								FB_MC2_AX5000_M_nMC_TouchProbe2_stTriggerInput.Edge:= Tc2_MC2.RisingEdge;
							END_IF
							FB_MC2_AX5000_M_nMC_TouchProbe2_fbTouchProbe(Axis:= _stAXIS_REF, TriggerInput:= FB_MC2_AX5000_M_nMC_TouchProbe2_stTriggerInput, Execute:= FALSE, WindowOnly:= FALSE);
						END_IF
					END_IF	
				END_IF			
				
			ELSE
				FB_MC2_AX5000_M_nMC_TouchProbe2_iState:= 000;
			END_IF
			
ELSE
	FB_MC2_AX5000_M_nMC_TouchProbe2_iState:= 000;
END_CASE
END_METHOD

//	The result of the method is an unsigned double integer
//	0 = idle 
//	1 = coupled
//	2 = starting
//	3 = running
//	4 = aborted
// 	5 = no hardware connected
// 	6 = Spare
//	7 = pointer or index error
//	8 = mapping error
//	9 = parameter error
//	10 = complete
//	Any other number = ErrorID
METHOD PUBLIC M_nReset : UDINT
VAR_INPUT
	bExecute: BOOL;
END_VAR
//**********************************
// Wait for execute
//**********************************
FB_MC2_AX5000_M_nReset_fbExecute_R_TRIG(CLK:= bExecute);
IF FB_MC2_AX5000_M_nReset_fbExecute_R_TRIG.Q THEN
	FB_MC2_AX5000_M_nReset_fbSoEReset(Execute:= FALSE, Axis:= _stAXIS_REF); 
	SUPER^.M_nReset(bExecute:= FALSE);
	FB_MC2_AX5000_M_nReset_iState:= 001;
END_IF


//**********************************
// Main sequence
//**********************************
CASE FB_MC2_AX5000_M_nReset_iState OF

	000: 	// Do nothing

	001:	// Reset father	
			M_nReset:= Tc3_HBI_System.cRUNNING;
			FB_MC2_AX5000_M_nReset_nStatus:= SUPER^.M_nReset(bExecute:= TRUE); 
			IF FB_MC2_AX5000_M_nReset_nStatus = Tc3_HBI_System.cCOUPLED OR FB_MC2_AX5000_M_nReset_nStatus = Tc3_HBI_System.cCOMPLETE THEN		
				SUPER^.M_nReset(bExecute:= FALSE);
				FB_MC2_AX5000_M_nReset_fbSoEReset(Execute:= FALSE, Axis:= _stAXIS_REF); 
				IF _bHardwareConnected THEN
					FB_MC2_AX5000_M_nReset_iState:= FB_MC2_AX5000_M_nReset_iState +1;
				ELSE
					IF _stAXIS_REF.Status.Coupled THEN
						FB_MC2_AX5000_M_nReset_iState:= 020;
					ELSE
						FB_MC2_AX5000_M_nReset_iState:= 030;
					END_IF
				END_IF
			END_IF

	002:	// Reset AX5000
			M_nReset:= Tc3_HBI_System.cRUNNING;
			FB_MC2_AX5000_M_nReset_fbSoEReset(Execute:= TRUE, Axis:= _stAXIS_REF); 
			
			// Error handling
			IF FB_MC2_AX5000_M_nReset_fbSoEReset.Error THEN
				M_nError(FB_MC2_AX5000_M_nReset_fbSoEReset.AdsErrId);
				M_nReset:= FB_MC2_AX5000_M_nReset_fbSoEReset.AdsErrId;
				IF _stAXIS_REF.Status.Coupled THEN
					FB_MC2_AX5000_M_nReset_iState:= 020;
				ELSE
					FB_MC2_AX5000_M_nReset_iState:= 030;
				END_IF	
			ELSE
				// Done
				IF NOT FB_MC2_AX5000_M_nReset_fbSoEReset.Busy THEN
					IF _stAXIS_REF.Status.Coupled THEN
						FB_MC2_AX5000_M_nReset_iState:= 020;
					ELSE
						FB_MC2_AX5000_M_nReset_iState:= 030;
					END_IF	
				END_IF	
			END_IF

	020:	// Coupled
			M_nReset:= Tc3_HBI_System.cCOUPLED;
			IF NOT bExecute THEN
				FB_MC2_AX5000_M_nReset_fbSoEReset(Execute:= FALSE, Axis:= _stAXIS_REF); 
				SUPER^.M_nReset(bExecute:= FALSE);
				FB_MC2_AX5000_M_nReset_iState:= 000;
			END_IF	

	030: 	// Done
			M_nReset:= Tc3_HBI_System.cCOMPLETE;
			IF NOT bExecute THEN
				FB_MC2_AX5000_M_nReset_fbSoEReset(Execute:= FALSE, Axis:= _stAXIS_REF); 
				SUPER^.M_nReset(bExecute:= FALSE);
				FB_MC2_AX5000_M_nReset_iState:= 000;
			END_IF	
		
ELSE
	FB_MC2_AX5000_M_nReset_iState:= 000;
END_CASE
END_METHOD

PROPERTY PUBLIC P_lrRecordedPosition1_RisingEdge : LREAL
GET
P_lrRecordedPosition1_RisingEdge:= FB_MC2_AX5000_M_nMC_TouchProbe1_lrRecordedPosition1_RisingEdge;
END_GET
END_PROPERTY

PROPERTY PUBLIC P_lrRecordedPosition2_FallingEdge : LREAL
GET
P_lrRecordedPosition2_FallingEdge:= FB_MC2_AX5000_M_nMC_TouchProbe2_lrRecordedPosition2_FallingEdge;
END_GET
END_PROPERTY

PROPERTY PUBLIC P_lrRecordedPosition2_RisingEdge : LREAL
GET
P_lrRecordedPosition2_RisingEdge:= FB_MC2_AX5000_M_nMC_TouchProbe2_lrRecordedPosition2_RisingEdge;
END_GET
END_PROPERTY

PROPERTY PUBLIC P_nDiagnosticNumber : UDINT
GET
P_nDiagnosticNumber:= FB_MC2_AX5000_M_nMC_DriveData_nDiagnosticNumber;
END_GET
END_PROPERTY

PROPERTY PUBLIC P_rActualMainVoltage : REAL
GET
P_rActualMainVoltage:= LREAL_TO_REAL(FB_MC2_AX5000_M_nMC_DriveData_lrActualMainVoltage);
END_GET
END_PROPERTY

PROPERTY PUBLIC P_rAmplifierTemperature : REAL
GET
P_rAmplifierTemperature:= LREAL_TO_REAL(FB_MC2_AX5000_M_nMC_DriveData_lrAmplifierTemperature);
END_GET
END_PROPERTY

PROPERTY PUBLIC P_rMotorTemperature : REAL
GET
P_rMotorTemperature:= LREAL_TO_REAL(FB_MC2_AX5000_M_nMC_DriveData_lrMotorTemperature);
END_GET
END_PROPERTY

PROPERTY PUBLIC P_sDiagnosticNumber : STRING
GET
P_sDiagnosticNumber:= Tc2_Utilities.DWORD_TO_HEXSTR( FB_MC2_AX5000_M_nMC_DriveData_nDiagnosticNumber, 4, FALSE );
END_GET
END_PROPERTY

END_FUNCTION_BLOCK

// MOTION/POUs/FBs/Basic/FB_MC2_Basic
//------------------------------------------------------------------------------------------
//                                                                                        	
//***************************** Beckhoff TwinCAT Examples **********************************
//                                                                                        	
//************************************* WARNING ********************************************
// This program is only an example. If it is used as a control program in any real        	
// application, Beckhoff is not responsible for any malfunction, loss or damage           	
// which could arise by using this program!                                               	
//                                                                                        	
//*************************************  Program Info. *************************************
//                                                                                        	
// PLC program name:       	FB_MC2_AxisBasic (FB)                                          	
// Hardware platform:      	TwinCat PTP v3.1.4022				                          	                                  	
//                                                                                        	
// ======================================================================================== 
//         Version       Date                        Remarks                              	
// ======================================================================================== 
//         3.1           27 feb 2018                 First release of this example    
//         3.7.1.1		 09 may 2018    			 Next release of this example
// ======================================================================================== 
//                                                                                        	
//******************************* Aims OF this PLC PROGRAM *********************************
//                                                                                        	
// MC2 servo axis 						 			                                      	
// Add axis error message 																	                      	
//                                                                                        	
//----------------------------------------------------------------------------------------- 
FUNCTION_BLOCK FB_MC2_Basic EXTENDS FB_MC2_Compact IMPLEMENTS I_MC2_Basic
VAR
//***************************
// Metods variable
//***************************
	FB_MC2_AxisBasic_M_nMC_ClrLagError_bExecute: BOOL;
	FB_MC2_AxisBasic_M_nMC_ClrLagError_iState: INT;
	FB_MC2_AxisBasic_M_nMC_ClrLagError_fbExecute_R_TRIG: Tc2_Standard.R_TRIG;
	FB_MC2_AxisBasic_M_nMC_ClrLagError_stSetPositionOptions: Tc2_MC2.ST_SetPositionOptions;
	FB_MC2_AxisBasic_M_nMC_ClrLagError_fbSetPositon: Tc2_MC2.MC_SetPosition;
	
	FB_MC2_AxisBasic_M_nMC_DeadTimeComp_iState: INT;
	FB_MC2_AxisBasic_M_nMC_DeadTimeComp_fbADSREAD: TC2_SYSTEM.ADSREAD;
	FB_MC2_AxisBasic_M_nMC_DeadTimeComp_fbADSWRITE: TC2_SYSTEM.ADSWRITE;
	FB_MC2_AxisBasic_M_nMC_DeadTimeComp_nAxisCycleTime: UDINT;
	FB_MC2_AxisBasic_M_nMC_DeadTimeComp_lrDeadTimeComp: LREAL;
	
	FB_MC2_AxisBasic_M_nMC_GearIn_bExecute: BOOL;
	FB_MC2_AxisBasic_M_nMC_GearIn_pMaster: POINTER TO TC2_MC2.AXIS_REF;
	FB_MC2_AxisBasic_M_nMC_GearIn_lrRatioNumerator: LREAL;
	FB_MC2_AxisBasic_M_nMC_GearIn_iRatioDenominator: UINT;
	FB_MC2_AxisBasic_M_nMC_GearIn_fbMC2_GearIn: TC2_MC2.MC_GearIn;

	FB_MC2_AxisBasic_M_nMC_GearInDyn_bEnable: BOOL;
	FB_MC2_AxisBasic_M_nMC_GearInDyn_pMaster: POINTER TO TC2_MC2.AXIS_REF;
	FB_MC2_AxisBasic_M_nMC_GearInDyn_lrGearRatio: LREAL;
	FB_MC2_AxisBasic_M_nMC_GearInDyn_fbMC2_GearInDyn: TC2_MC2.MC_GearInDyn;

	FB_MC2_AxisBasic_M_nMC_GearInMultiMaster_bEnable: BOOL;
	FB_MC2_AxisBasic_M_nMC_GearInMultiMaster_pMaster1: POINTER TO Tc2_MC2.AXIS_REF;
	FB_MC2_AxisBasic_M_nMC_GearInMultiMaster_pMaster2: POINTER TO Tc2_MC2.AXIS_REF;
	FB_MC2_AxisBasic_M_nMC_GearInMultiMaster_pMaster3: POINTER TO Tc2_MC2.AXIS_REF;
	FB_MC2_AxisBasic_M_nMC_GearInMultiMaster_pMaster4: POINTER TO Tc2_MC2.AXIS_REF;
	FB_MC2_AxisBasic_M_nMC_GearInMultiMaster_bAdvancedSlaveDynamics: BOOL;
	FB_MC2_AxisBasic_M_nMC_GearInMultiMaster_lrGearRatio1: LREAL;
	FB_MC2_AxisBasic_M_nMC_GearInMultiMaster_lrGearRatio2: LREAL;
	FB_MC2_AxisBasic_M_nMC_GearInMultiMaster_lrGearRatio3: LREAL;
	FB_MC2_AxisBasic_M_nMC_GearInMultiMaster_lrGearRatio4: LREAL;
	FB_MC2_AxisBasic_M_nMC_GearInMultiMaster_fbMC_GearInMultiMaster: Tc2_MC2.MC_GearInMultiMaster;

	FB_MC2_AxisBasic_M_nMC_GearOut_bExecute: BOOL;
	FB_MC2_AxisBasic_M_nMC_GearOut_fbMC2_GearOut: TC2_MC2.MC_GearOut;

	FB_MC2_AxisBasic_M_nMC_InverseMotor_bExecute: BOOL;
	FB_MC2_AxisBasic_M_nMC_InverseMotor_bInverse: BOOL;
	FB_MC2_AxisBasic_M_nMC_InverseMotor_iState: INT;
	FB_MC2_AxisBasic_M_nMC_InverseMotor_fbExecute_R_TRIG: Tc2_Standard.R_TRIG;
	FB_MC2_AxisBasic_M_nMC_InverseMotor_fbADSRDWRT: Tc2_System.ADSRDWRT;
	FB_MC2_AxisBasic_M_nMC_InverseMotor_stMC2_Param: _ST_MC2_Param2;
	FB_MC2_AxisBasic_M_nMC_InverseMotor_arr_nADSReturn: ARRAY[1..4] OF UDINT;

	FB_MC2_AxisBasic_M_nMC_PhasingAbsolute_bExecute: BOOL;
	FB_MC2_AxisBasic_M_nMC_PhasingAbsolute_pMaster: POINTER TO TC2_MC2.AXIS_REF;
	FB_MC2_AxisBasic_M_nMC_PhasingAbsolute_lrPhaseShift: LREAL;
	FB_MC2_AxisBasic_M_nMC_PhasingAbsolute_lrVelocity: LREAL;
	FB_MC2_AxisBasic_M_nMC_PhasingAbsolute_lrAbsolutePhaseShift: LREAL;
	FB_MC2_AxisBasic_M_nMC_PhasingAbsolute_iState: INT;
	FB_MC2_AxisBasic_M_nMC_PhasingAbsolute_fbExecute_R_TRIG: R_TRIG;
	FB_MC2_AxisBasic_M_nMC_PhasingAbsolute_fbNotExecute_R_TRIG: R_TRIG;
	FB_MC2_AxisBasic_M_nMC_PhasingAbsolute_fbMC2_HaltParsing: Tc2_MC2.MC_HaltPhasing;
	FB_MC2_AxisBasic_M_nMC_PhasingAbsolute_fbMC2_PhasingAbsolute: Tc2_MC2.MC_PhasingAbsolute;
	
	FB_MC2_AxisBasic_M_nMC_PhasingRelative_bExecute: BOOL;
	FB_MC2_AxisBasic_M_nMC_PhasingRelative_pMaster: POINTER TO TC2_MC2.AXIS_REF;
	FB_MC2_AxisBasic_M_nMC_PhasingRelative_lrPhaseShift: LREAL;
	FB_MC2_AxisBasic_M_nMC_PhasingRelative_lrVelocity: LREAL;
	FB_MC2_AxisBasic_M_nMC_PhasingRelative_lrCoveredPhaseShift: LREAL;
	FB_MC2_AxisBasic_M_nMC_PhasingRelative_iState: INT;
	FB_MC2_AxisBasic_M_nMC_PhasingRelative_fbExecute_R_TRIG: R_TRIG;
	FB_MC2_AxisBasic_M_nMC_PhasingRelative_fbNotExecute_R_TRIG: R_TRIG;
	FB_MC2_AxisBasic_M_nMC_PhasingRelative_fbMC2_HaltParsing: Tc2_MC2.MC_HaltPhasing;
	FB_MC2_AxisBasic_M_nMC_PhasingRelative_fbMC2_PhasingRelative: Tc2_MC2.MC_PhasingRelative;

	FB_MC2_AxisBasic_M_nMC_PositionLagMonitoring_bEnable: BOOL;
	FB_MC2_AxisBasic_M_nMC_PositionLagMonitoring_bDisable: BOOL;
	FB_MC2_AxisBasic_M_nMC_PositionLagMonitoring_iState: INT;
	FB_MC2_AxisBasic_M_nMC_PositionLagMonitoring_fbExecute1_R_TRIG: Tc2_Standard.R_TRIG;
	FB_MC2_AxisBasic_M_nMC_PositionLagMonitoring_fbExecute2_R_TRIG: Tc2_Standard.R_TRIG;
	FB_MC2_AxisBasic_M_nMC_PositionLagMonitoring_fbADSWrite: Tc2_System.ADSWRITE;
	FB_MC2_AxisBasic_M_nMC_PositionLagMonitoring_nData: UINT;

	FB_MC2_AxisBasic_M_nMC_Power_bEnable: BOOL;
	FB_MC2_AxisBasic_M_nMC_Power_bE_Stop: BOOL;
	FB_MC2_AxisBasic_M_nMC_Power_bE_StopDelay: BOOL;
	FB_MC2_AxisBasic_M_nMC_Power_bEnable_Positive: BOOL;
	FB_MC2_AxisBasic_M_nMC_Power_bEnable_Negative: BOOL; 
	FB_MC2_AxisBasic_M_nMC_Power_Status: UDINT;

	FB_MC2_AxisBasic_M_nMC_ReadParameter_iState: INT;
	FB_MC2_AxisBasic_M_nMC_ReadParameter_bDone: BOOL;
	FB_MC2_AxisBasic_M_nMC_ReadParameter_lrTempMaxVelocity: LREAL;
	FB_MC2_AxisBasic_M_nMC_ReadParameter_lrMaxVelocity: LREAL;
	FB_MC2_AxisBasic_M_nMC_ReadParameter_fbExecute_R_TRIG: Tc2_Standard.R_TRIG;
	FB_MC2_AxisBasic_M_nMC_ReadParameter_fbADSREAD	: Tc2_System.ADSREAD;
	
	FB_MC2_AxisBasic_M_nMC_RegCorrectiom_bExecute: BOOL;
	FB_MC2_AxisBasic_M_nMC_RegCorrectiom_pRegCorrection: POINTER TO ST_MC2_RegCorrection;
	FB_MC2_AxisBasic_M_nMC_RegCorrectiom_iState: INT;
	FB_MC2_AxisBasic_M_nMC_RegCorrectiom_fbExecute_R_TRIG: R_TRIG;
	FB_MC2_AxisBasic_M_nMC_RegCorrectiom_fbNotExecute_R_TRIG: R_TRIG;
	FB_MC2_AxisBasic_M_nMC_RegCorrectiom_fbMC2_AbortSuperposition : Tc2_MC2.MC_AbortSuperposition;
	FB_MC2_AxisBasic_M_nMC_RegCorrectiom_fbMC2_MoveSuperImposed : Tc2_MC2.MC_MoveSuperImposed;

	FB_MC2_AxisBasic_M_nMC_SetEncoderOffset_bExecute: BOOL;
	FB_MC2_AxisBasic_M_nMC_SetEncoderOffset_lrOffset: LREAL;
	FB_MC2_AxisBasic_M_nMC_SetEncoderOffset_iState: INT;
	FB_MC2_AxisBasic_M_nMC_SetEncoderOffset_fbExecute_R_TRIG: Tc2_Standard.R_TRIG;
	FB_MC2_AxisBasic_M_nMC_SetEncoderOffset_fbADSWRITE	: ADSWRITE;
	
	FB_MC2_AxisBasic_M_nMC_SetFeedConstant_bExecute: BOOL;
	FB_MC2_AxisBasic_M_nMC_SetFeedConstant_lrFeedConstant: LREAL;
	FB_MC2_AxisBasic_M_nMC_SetFeedConstant_iState: INT;
	FB_MC2_AxisBasic_M_nMC_SetFeedConstant_fbExecute_R_TRIG: Tc2_Standard.R_TRIG;
	FB_MC2_AxisBasic_M_nMC_SetFeedConstant_fbADSWRITE	: ADSWRITE;
	
	FB_MC2_AxisBasic_M_nMC_SetModuloFactor_bExecute: BOOL;
	FB_MC2_AxisBasic_M_nMC_SetModuloFactor_lrModuloFactor: LREAL;
	FB_MC2_AxisBasic_M_nMC_SetModuloFactor_iState: INT;
	FB_MC2_AxisBasic_M_nMC_SetModuloFactor_fbExecute_R_TRIG: Tc2_Standard.R_TRIG;
	FB_MC2_AxisBasic_M_nMC_SetModuloFactor_fbADSWRITE: TC2_SYSTEM.ADSWRITE;
	
	FB_MC2_AxisBasic_M_nMC_SetPosition_bExecute: BOOL;
	FB_MC2_AxisBasic_M_nMC_SetPosition_lrPosition: LREAL;
	FB_MC2_AxisBasic_M_nMC_SetPosition_iState: INT;
	FB_MC2_AxisBasic_M_nMC_SetPosition_fbExecute_R_TRIG: Tc2_Standard.R_TRIG;
	FB_MC2_AxisBasic_M_nMC_SetPosition_fbMC2_SetPosition: Tc2_MC2.MC_SetPosition;

	FB_MC2_AxisBasic_M_nMC_SetPositionRelative_bExecute: BOOL;
	FB_MC2_AxisBasic_M_nMC_SetPositionRelative_lrPosition: LREAL;
	FB_MC2_AxisBasic_M_nMC_SetPositionRelative_iState: INT;
	FB_MC2_AxisBasic_M_nMC_SetPositionRelative_fbExecute_R_TRIG: Tc2_Standard.R_TRIG;
	FB_MC2_AxisBasic_M_nMC_SetPositionRelative_fbMC2_SetPosition: Tc2_MC2.MC_SetPosition;

	FB_MC2_AxisBasic_M_nMC_SetScaleFactor_bExecute: BOOL;
	FB_MC2_AxisBasic_M_nMC_SetScaleFactor_lrScaleFactor: LREAL;
	FB_MC2_AxisBasic_M_nMC_SetScaleFactor_iState: INT;
	FB_MC2_AxisBasic_M_nMC_SetScaleFactor_fbExecute_R_TRIG: Tc2_Standard.R_TRIG;
	FB_MC2_AxisBasic_M_nMC_SetScaleFactor_fbMC2_SetEncoderScalingFactor: Tc2_MC2.MC_SetEncoderScalingFactor;

	FB_MC2_AxisBasic_M_nMC_SetVeloKvFactor_bExecute: BOOL;
	FB_MC2_AxisBasic_M_nMC_SetVeloKvFactor_lrKvFactor: LREAL;
	FB_MC2_AxisBasic_M_nMC_SetVeloKvFactor_iState: INT;
	FB_MC2_AxisBasic_M_nMC_SetVeloKvFactor_fbExecute_R_TRIG: Tc2_Standard.R_TRIG;
	FB_MC2_AxisBasic_M_nMC_SetVeloKvFactor_fbADSWRITE: TC2_SYSTEM.ADSWRITE;
	
	FB_MC2_AxisBasic_M_nReset_bExecute: BOOL;
	FB_MC2_AxisBasic_M_nReset_bError: BOOL;
	FB_MC2_AxisBasic_M_nReset_iState: INT;
	FB_MC2_AxisBasic_M_nReset_fbExecute_R_TRIG: Tc2_Standard.R_TRIG;
	FB_MC2_AxisBasic_M_nReset_fbMC2_Reset: Tc2_MC2.MC_Reset;
	FB_MC2_AxisBasic_M_nReset_nStatus: UDINT;
END_VAR

//	The result of the method is an unsigned double integer
//	0 = idle 
//	1 = coupled
//	2 = starting
//	3 = running
//	4 = aborted
// 	5 = no hardware connected
// 	6 = Spare
//	7 = pointer or index error
//	8 = mapping error
//	9 = parameter error
//	10 = complete
//	Any other number = ErrorID
METHOD PUBLIC M_nMC_ClrLagError : UDINT
VAR_INPUT
	bExecute: BOOL;
END_VAR
// Local variable
FB_MC2_AxisBasic_M_nMC_ClrLagError_bExecute:= bExecute;

//**********************************
// Reset 
//**********************************
IF _bReset THEN
	IF _bError THEN
		FB_MC2_AxisBasic_M_nMC_ClrLagError_fbSetPositon(Axis:= _stAXIS_REF, Execute:= FALSE); 
		FB_MC2_AxisBasic_M_nMC_ClrLagError_iState:= 000;
	END_IF
END_IF

//**********************************
// Wait for execute
//**********************************
IF _stAXIS_REF.NcToPlc.AxisID > 0 THEN
	FB_MC2_AxisBasic_M_nMC_ClrLagError_fbExecute_R_TRIG(CLK:= FB_MC2_AxisBasic_M_nMC_ClrLagError_bExecute);
	IF FB_MC2_AxisBasic_M_nMC_ClrLagError_fbExecute_R_TRIG.Q THEN
		FB_MC2_AxisBasic_M_nMC_ClrLagError_fbSetPositon(Axis:= _stAXIS_REF, Execute:= FALSE); 
		FB_MC2_AxisBasic_M_nMC_ClrLagError_iState:= 001;
	END_IF
ELSE
	FB_MC2_AxisBasic_M_nMC_ClrLagError_fbExecute_R_TRIG(CLK:= FALSE);
	FB_MC2_AxisBasic_M_nMC_ClrLagError_iState:= 000;
	IF FB_MC2_AxisBasic_M_nMC_ClrLagError_bExecute THEN
		M_nMC_ClrLagError:= Tc3_HBI_System.cMAPPING_ERROR;
	END_IF
	RETURN;
END_IF


//**********************************
// Main sequence
//**********************************
CASE FB_MC2_AxisBasic_M_nMC_ClrLagError_iState OF

	000: 	// Do nothing

	001:	// Reset lag error
			M_nMC_ClrLagError:= Tc3_HBI_System.cSTARTING;
			FB_MC2_AxisBasic_M_nMC_ClrLagError_stSetPositionOptions.ClearPositionLag:= TRUE;
			FB_MC2_AxisBasic_M_nMC_ClrLagError_fbSetPositon(
				Axis:= _stAXIS_REF, 
				Execute:= TRUE, 
				Position:= _stAXIS_REF.NcToPlc.ActPos, 
				Mode:= , 
				Options:= FB_MC2_AxisBasic_M_nMC_ClrLagError_stSetPositionOptions, 
				Done=> , 
				Busy=> , 
				Error=> , 
				ErrorID=> );

			// Error handling
			IF FB_MC2_AxisBasic_M_nMC_ClrLagError_fbSetPositon.Error THEN
				M_nError(nErrorID:= FB_MC2_AxisBasic_M_nMC_ClrLagError_fbSetPositon.ErrorID);
				M_nMC_ClrLagError:= FB_MC2_AxisBasic_M_nMC_ClrLagError_fbSetPositon.ErrorID;
			ELSE
				// Done
				IF FB_MC2_AxisBasic_M_nMC_ClrLagError_fbSetPositon.Done THEN
					FB_MC2_AxisBasic_M_nMC_ClrLagError_iState:= FB_MC2_AxisBasic_M_nMC_ClrLagError_iState +1;
				END_IF
			END_IF

	002:	// Done
			M_nMC_ClrLagError:= Tc3_HBI_System.cCOMPLETE;
			IF NOT FB_MC2_AxisBasic_M_nMC_ClrLagError_bExecute THEN
				FB_MC2_AxisBasic_M_nMC_ClrLagError_fbSetPositon(Axis:= _stAXIS_REF, Execute:= FALSE); 
				FB_MC2_AxisBasic_M_nMC_ClrLagError_iState:= 000;
			END_IF

ELSE
	FB_MC2_AxisBasic_M_nMC_ClrLagError_iState:= 000;
END_CASE
END_METHOD

//	The result of the method is an unsigned double integer
//	0 = idle 
//	1 = coupled
//	2 = starting
//	3 = running
//	4 = aborted
// 	5 = no hardware connected
// 	6 = Spare
//	7 = pointer or index error
//	8 = mapping error
//	9 = parameter error
//	10 = complete
//	Any other number = ErrorID
METHOD PUBLIC M_nMC_DeadTimeComp : UDINT
//**********************************
// Reset 
//**********************************
IF _bReset THEN
	FB_MC2_AxisBasic_M_nMC_DeadTimeComp_fbADSREAD(READ:= FALSE);
	FB_MC2_AxisBasic_M_nMC_DeadTimeComp_iState:= 000;
ELSE
	// No hardware connected
	IF NOT _bHardwareConnected THEN
		FB_MC2_AxisBasic_M_nMC_DeadTimeComp_iState:= 000;
		M_nMC_DeadTimeComp:= Tc3_HBI_System.cNO_HARDWARE_CONNECTED;
		RETURN;
	END_IF
END_IF

// Check for Axis
IF _stAXIS_REF.NcToPlc.AxisID = 0 THEN
	FB_MC2_AxisBasic_M_nMC_DeadTimeComp_iState:= 000;
	RETURN;
END_IF


//**********************************
// Main sequence
//**********************************
CASE FB_MC2_AxisBasic_M_nMC_DeadTimeComp_iState OF

	000:	// Init
			FB_MC2_AxisBasic_M_nMC_DeadTimeComp_fbADSREAD(READ:= FALSE);
			IF _stAXIS_REF.NcToPlc.AxisID > 0 THEN
				IF FB_MC2_AxisBasic_M_nMC_DeadTimeComp_nAxisCycleTime > 0 THEN
					FB_MC2_AxisBasic_M_nMC_DeadTimeComp_iState:= 010;
				ELSE
					FB_MC2_AxisBasic_M_nMC_DeadTimeComp_iState:= FB_MC2_AxisBasic_M_nMC_DeadTimeComp_iState +1;
				END_IF
			END_IF
	
	001:	// Read axis cycle time
			M_nMC_DeadTimeComp:= Tc3_HBI_System.cSTARTING;
			FB_MC2_AxisBasic_M_nMC_DeadTimeComp_fbADSREAD(READ:= FALSE);
			FB_MC2_AxisBasic_M_nMC_DeadTimeComp_fbADSREAD(
				NETID:= '', 
				PORT:= AMSPORT_R0_NC, 
				IDXGRP:= 16#4000 + _stAXIS_REF.NcToPlc.AxisId, 
				IDXOFFS:= 16#0004, 
				LEN:= SIZEOF(FB_MC2_AxisBasic_M_nMC_DeadTimeComp_nAxisCycleTime), 
				DESTADDR:= ADR(FB_MC2_AxisBasic_M_nMC_DeadTimeComp_nAxisCycleTime), 
				READ:= TRUE); 
		
			FB_MC2_AxisBasic_M_nMC_DeadTimeComp_iState:= FB_MC2_AxisBasic_M_nMC_DeadTimeComp_iState +1;

	002:	// Read done	
			M_nMC_DeadTimeComp:= Tc3_HBI_System.cRUNNING;
			FB_MC2_AxisBasic_M_nMC_DeadTimeComp_fbADSREAD(READ:= TRUE);
	
			// Error
			IF FB_MC2_AxisBasic_M_nMC_DeadTimeComp_fbADSREAD.ERR THEN
				M_nError(nErrorID:= FB_MC2_AxisBasic_M_nMC_DeadTimeComp_fbADSREAD.ERRID);
				M_nMC_DeadTimeComp:= FB_MC2_AxisBasic_M_nMC_DeadTimeComp_fbADSREAD.ERRID;
			ELSE
				// Done
				IF NOT FB_MC2_AxisBasic_M_nMC_DeadTimeComp_fbADSREAD.BUSY THEN
					FB_MC2_AxisBasic_M_nMC_DeadTimeComp_fbADSREAD(READ:= FALSE);
					FB_MC2_AxisBasic_M_nMC_DeadTimeComp_iState:= FB_MC2_AxisBasic_M_nMC_DeadTimeComp_iState +1;
				END_IF
			END_IF

	003:	// Write dead time compensation to axis parameter
			M_nMC_DeadTimeComp:= Tc3_HBI_System.cRUNNING;
			FB_MC2_AxisBasic_M_nMC_DeadTimeComp_lrDeadTimeComp:= (UDINT_TO_LREAL(FB_MC2_AxisBasic_M_nMC_DeadTimeComp_nAxisCycleTime) / 1000000.0) * 4.0; 
			FB_MC2_AxisBasic_M_nMC_DeadTimeComp_fbADSWRITE(WRITE:= FALSE); 
			FB_MC2_AxisBasic_M_nMC_DeadTimeComp_fbADSWRITE(
				NETID:= '', 
				PORT:= AMSPORT_R0_NC, 
				IDXGRP:= 16#4000 + _stAXIS_REF.NcToPlc.AxisId, 
				IDXOFFS:= 16#0104, 
				LEN:= SIZEOF(FB_MC2_AxisBasic_M_nMC_DeadTimeComp_lrDeadTimeComp), 
				SRCADDR:= ADR(FB_MC2_AxisBasic_M_nMC_DeadTimeComp_lrDeadTimeComp), 
				WRITE:= TRUE); 
	
			FB_MC2_AxisBasic_M_nMC_DeadTimeComp_iState:= FB_MC2_AxisBasic_M_nMC_DeadTimeComp_iState +1;
				
	004:	// Write done	
			M_nMC_DeadTimeComp:= Tc3_HBI_System.cRUNNING;
			FB_MC2_AxisBasic_M_nMC_DeadTimeComp_fbADSWRITE(WRITE:= TRUE); 
	
			// Error
			IF FB_MC2_AxisBasic_M_nMC_DeadTimeComp_fbADSWRITE.ERR THEN
				M_nError(nErrorID:= FB_MC2_AxisBasic_M_nMC_DeadTimeComp_fbADSWRITE.ERRID);
				M_nMC_DeadTimeComp:= FB_MC2_AxisBasic_M_nMC_DeadTimeComp_fbADSWRITE.ERRID;
			ELSE
				// Done
				IF NOT FB_MC2_AxisBasic_M_nMC_DeadTimeComp_fbADSWRITE.BUSY THEN
					FB_MC2_AxisBasic_M_nMC_DeadTimeComp_fbADSWRITE(WRITE:= FALSE); 
					FB_MC2_AxisBasic_M_nMC_DeadTimeComp_iState:= 10;
				END_IF
			END_IF
	
	010:	// Done
		M_nMC_DeadTimeComp:= Tc3_HBI_System.cCOMPLETE;
	
ELSE
	FB_MC2_AxisBasic_M_nMC_DeadTimeComp_iState:= 000;
END_CASE
END_METHOD

//	The result of the method is an unsigned double integer
//	0 = idle 
//	1 = coupled
//	2 = starting
//	3 = running
//	4 = aborted
// 	5 = no hardware connected
// 	6 = Spare
//	7 = pointer or index error
//	8 = mapping error
//	9 = parameter error
//	10 = complete
//	Any other number = ErrorID
METHOD PUBLIC M_nMC_GearIn : UDINT
VAR_INPUT
	bExecute: BOOL;
	pMaster: POINTER TO TC2_MC2.AXIS_REF;
	lrRatioNumerator: LREAL;
	iRatioDenominator: UINT;
END_VAR
// Local variable
FB_MC2_AxisBasic_M_nMC_GearIn_bExecute:= bExecute;
FB_MC2_AxisBasic_M_nMC_GearIn_pMaster:= pMaster;
FB_MC2_AxisBasic_M_nMC_GearIn_lrRatioNumerator:= lrRatioNumerator;
FB_MC2_AxisBasic_M_nMC_GearIn_iRatioDenominator:= iRatioDenominator;

//****************************
// Pointer and axis id check 
//****************************
IF _stAXIS_REF.NcToPlc.AxisID > 0 THEN
	// Pointer check
	IF FB_MC2_AxisBasic_M_nMC_GearIn_pMaster = 0 THEN
		M_nMC_GearIn:= Tc3_HBI_System.cPOINTER_OR_INDEX_ERROR;
		RETURN;
	ELSE	
		// Reset
		IF _bReset THEN
			IF FB_MC2_AxisBasic_M_nMC_GearIn_fbMC2_GearIn.Error THEN
				// Gear in
				FB_MC2_AxisBasic_M_nMC_GearIn_fbMC2_GearIn(
					Master:= FB_MC2_AxisBasic_M_nMC_GearIn_pMaster^, 
					Slave:= _stAXIS_REF, 
					Execute:= FALSE, 
					RatioNumerator:= FB_MC2_AxisBasic_M_nMC_GearIn_lrRatioNumerator, 
					RatioDenominator:= FB_MC2_AxisBasic_M_nMC_GearIn_iRatioDenominator, 
					Acceleration:= _stDynamic.lrAcceleration, 
					Deceleration:= _stDynamic.lrDeceleration, 
					Jerk:= _stDynamic.lrJerk, 
					BufferMode:= , 
					Options:= , 
					InGear=> , 
					Busy=> , 
					Active=> , 
					CommandAborted=> , 
					Error=> , 
					ErrorID=> );
			ELSE
				// Gear in
				FB_MC2_AxisBasic_M_nMC_GearIn_fbMC2_GearIn(
					Master:= FB_MC2_AxisBasic_M_nMC_GearIn_pMaster^, 
					Slave:= _stAXIS_REF, 
					Execute:= FB_MC2_AxisBasic_M_nMC_GearIn_bExecute, 
					RatioNumerator:= FB_MC2_AxisBasic_M_nMC_GearIn_lrRatioNumerator, 
					RatioDenominator:= FB_MC2_AxisBasic_M_nMC_GearIn_iRatioDenominator, 
					Acceleration:= _stDynamic.lrAcceleration, 
					Deceleration:= _stDynamic.lrDeceleration, 
					Jerk:= _stDynamic.lrJerk, 
					BufferMode:= , 
					Options:= , 
					InGear=> , 
					Busy=> , 
					Active=> , 
					CommandAborted=> , 
					Error=> , 
					ErrorID=> );
			END_IF	
		ELSE
			// Gear in
			FB_MC2_AxisBasic_M_nMC_GearIn_fbMC2_GearIn(
				Master:= FB_MC2_AxisBasic_M_nMC_GearIn_pMaster^, 
				Slave:= _stAXIS_REF, 
				Execute:= FB_MC2_AxisBasic_M_nMC_GearIn_bExecute, 
				RatioNumerator:= FB_MC2_AxisBasic_M_nMC_GearIn_lrRatioNumerator, 
				RatioDenominator:= FB_MC2_AxisBasic_M_nMC_GearIn_iRatioDenominator, 
				Acceleration:= _stDynamic.lrAcceleration, 
				Deceleration:= _stDynamic.lrDeceleration, 
				Jerk:= _stDynamic.lrJerk, 
				BufferMode:= , 
				Options:= , 
				InGear=> , 
				Busy=> , 
				Active=> , 
				CommandAborted=> , 
				Error=> , 
				ErrorID=> );
		END_IF
		
		// Error	
		IF FB_MC2_AxisBasic_M_nMC_GearIn_fbMC2_GearIn.Error THEN
			M_nError(nErrorID:= FB_MC2_AxisBasic_M_nMC_GearIn_fbMC2_GearIn.ErrorID);
			M_nMC_GearIn:= FB_MC2_AxisBasic_M_nMC_GearIn_fbMC2_GearIn.ErrorID;
		ELSE
			// Done
			IF FB_MC2_AxisBasic_M_nMC_GearIn_fbMC2_GearIn.CommandAborted THEN
				M_nMC_GearIn:= Tc3_HBI_System.cABORTED;
			ELSE
				IF FB_MC2_AxisBasic_M_nMC_GearIn_bExecute THEN
					IF FB_MC2_AxisBasic_M_nMC_GearIn_fbMC2_GearIn.InGear AND _stAXIS_REF.Status.Coupled THEN
						M_nMC_GearIn:= Tc3_HBI_System.cCOMPLETE;
					ELSE
						M_nMC_GearIn:= Tc3_HBI_System.cRUNNING;
					END_IF
				ELSE
					M_nMC_GearIn:= Tc3_HBI_System.cIDLE;
				END_IF
			END_IF
		END_IF		
	END_IF
	
ELSE
	FB_MC2_AxisBasic_M_nMC_GearIn_fbMC2_GearIn(Master:= FB_MC2_AxisBasic_M_nMC_GearIn_pMaster^, Slave:= _stAXIS_REF, Execute:= FALSE); 
	IF FB_MC2_AxisBasic_M_nMC_GearIn_bExecute THEN
		M_nMC_GearIn:= Tc3_HBI_System.cMAPPING_ERROR;
	END_IF
	RETURN;
END_IF
END_METHOD

//	The result of the method is an unsigned double integer
//	0 = idle 
//	1 = coupled
//	2 = starting
//	3 = running
//	4 = aborted
// 	5 = no hardware
//	7 = pointer or index error
//	8 = mapping error
//	9 = parameter error
//	10 = complete
//	Any other number = ErrorID
METHOD PUBLIC M_nMC_GearInDyn : UDINT
VAR_INPUT
	bEnable: BOOL;
	pMaster: POINTER TO TC2_MC2.AXIS_REF;
	lrGearRatio: LREAL;
END_VAR
// Local variable
FB_MC2_AxisBasic_M_nMC_GearInDyn_bEnable:= bEnable;
FB_MC2_AxisBasic_M_nMC_GearInDyn_pMaster:= pMaster;
FB_MC2_AxisBasic_M_nMC_GearInDyn_lrGearRatio:= lrGearRatio;

//****************************
// Pointer and axis id check 
//****************************
IF _stAXIS_REF.NcToPlc.AxisID > 0 THEN
	// Pointer check
	IF FB_MC2_AxisBasic_M_nMC_GearInDyn_pMaster = 0 THEN
		M_nMC_GearInDyn:= Tc3_HBI_System.cPOINTER_OR_INDEX_ERROR;
		RETURN;
	ELSE
		// Reset
		IF _bReset THEN
			IF FB_MC2_AxisBasic_M_nMC_GearInDyn_fbMC2_GearInDyn.Error THEN
				// Gear in dyn
				FB_MC2_AxisBasic_M_nMC_GearInDyn_fbMC2_GearInDyn(
					Master:= FB_MC2_AxisBasic_M_nMC_GearInDyn_pMaster^, 
					Slave:= _stAXIS_REF, 
					Enable:= FALSE, 
					GearRatio:= FB_MC2_AxisBasic_M_nMC_GearInDyn_lrGearRatio, 
					Acceleration:= _stDynamic.lrAcceleration, 
					Deceleration:= _stDynamic.lrDeceleration, 
					Jerk:= _stDynamic.lrJerk, 
					BufferMode:= , 
					Options:= , 
					InGear=> , 
					Busy=> , 
					Active=> , 
					CommandAborted=> , 
					Error=> , 
					ErrorID=> );
			ELSE	
				// Gear in dyn
				FB_MC2_AxisBasic_M_nMC_GearInDyn_fbMC2_GearInDyn(
					Master:= FB_MC2_AxisBasic_M_nMC_GearInDyn_pMaster^, 
					Slave:= _stAXIS_REF, 
					Enable:= FB_MC2_AxisBasic_M_nMC_GearInDyn_bEnable, 
					GearRatio:= FB_MC2_AxisBasic_M_nMC_GearInDyn_lrGearRatio, 
					Acceleration:= _stDynamic.lrAcceleration, 
					Deceleration:= _stDynamic.lrDeceleration, 
					Jerk:= _stDynamic.lrJerk, 
					BufferMode:= , 
					Options:= , 
					InGear=> , 
					Busy=> , 
					Active=> , 
					CommandAborted=> , 
					Error=> , 
					ErrorID=> );
				END_IF
		ELSE
			// Gear in dyn
			FB_MC2_AxisBasic_M_nMC_GearInDyn_fbMC2_GearInDyn(
				Master:= FB_MC2_AxisBasic_M_nMC_GearInDyn_pMaster^, 
				Slave:= _stAXIS_REF, 
				Enable:= FB_MC2_AxisBasic_M_nMC_GearInDyn_bEnable, 
				GearRatio:= FB_MC2_AxisBasic_M_nMC_GearInDyn_lrGearRatio, 
				Acceleration:= _stDynamic.lrAcceleration, 
				Deceleration:= _stDynamic.lrDeceleration, 
				Jerk:= _stDynamic.lrJerk, 
				BufferMode:= , 
				Options:= , 
				InGear=> , 
				Busy=> , 
				Active=> , 
				CommandAborted=> , 
				Error=> , 
				ErrorID=> );
		END_IF
		
		// Error	
		IF FB_MC2_AxisBasic_M_nMC_GearInDyn_fbMC2_GearInDyn.Error THEN
			M_nError(nErrorID:= FB_MC2_AxisBasic_M_nMC_GearInDyn_fbMC2_GearInDyn.ErrorID);
			M_nMC_GearInDyn:= FB_MC2_AxisBasic_M_nMC_GearInDyn_fbMC2_GearInDyn.ErrorID;
		ELSE
			// Done
			IF FB_MC2_AxisBasic_M_nMC_GearInDyn_fbMC2_GearInDyn.CommandAborted THEN
				M_nMC_GearInDyn:= Tc3_HBI_System.cABORTED;
			ELSE
				IF FB_MC2_AxisBasic_M_nMC_GearInDyn_bEnable THEN
					IF FB_MC2_AxisBasic_M_nMC_GearInDyn_fbMC2_GearInDyn.InGear AND _stAXIS_REF.Status.Coupled THEN
						M_nMC_GearInDyn:= Tc3_HBI_System.cCOMPLETE;
					ELSE
						M_nMC_GearInDyn:= Tc3_HBI_System.cRUNNING;
					END_IF
				ELSE
					M_nMC_GearInDyn:= Tc3_HBI_System.cIDLE;
				END_IF
			END_IF
		END_IF
		
	END_IF
ELSE
	FB_MC2_AxisBasic_M_nMC_GearInDyn_fbMC2_GearInDyn(Master:= FB_MC2_AxisBasic_M_nMC_GearInDyn_pMaster^, Slave:= _stAXIS_REF, Enable:= FALSE); 
	IF FB_MC2_AxisBasic_M_nMC_GearInDyn_bEnable THEN
		M_nMC_GearInDyn:= Tc3_HBI_System.cMAPPING_ERROR;
	END_IF
	RETURN;
END_IF
END_METHOD

//	The result of the method is an unsigned double integer
//	0 = idle 
//	1 = coupled
//	2 = starting
//	3 = running
//	4 = aborted
// 	5 = no hardware connected
// 	6 = Spare
//	7 = pointer or index error
//	8 = mapping error
//	9 = parameter error
//	10 = complete
//	Any other number = ErrorID
METHOD PUBLIC M_nMC_GearInMultiMaster : UDINT
VAR_INPUT
	bEnable: BOOL;
	pMaster1: POINTER TO Tc2_MC2.AXIS_REF;
	pMaster2: POINTER TO Tc2_MC2.AXIS_REF;
	pMaster3: POINTER TO Tc2_MC2.AXIS_REF;
	pMaster4: POINTER TO Tc2_MC2.AXIS_REF;
END_VAR
// Local variable
FB_MC2_AxisBasic_M_nMC_GearInMultiMaster_bEnable:= bEnable;
FB_MC2_AxisBasic_M_nMC_GearInMultiMaster_pMaster1:= pMaster1;
FB_MC2_AxisBasic_M_nMC_GearInMultiMaster_pMaster2:= pMaster2;
FB_MC2_AxisBasic_M_nMC_GearInMultiMaster_pMaster3:= pMaster3;
FB_MC2_AxisBasic_M_nMC_GearInMultiMaster_pMaster4:= pMaster4;

//****************************
// Pointer and axis id check 
//****************************
IF _stAXIS_REF.NcToPlc.AxisID > 0 THEN
	// Pointer check
	IF FB_MC2_AxisBasic_M_nMC_GearInMultiMaster_pMaster1 = 0 OR FB_MC2_AxisBasic_M_nMC_GearInMultiMaster_pMaster2 = 0 OR FB_MC2_AxisBasic_M_nMC_GearInMultiMaster_pMaster3 = 0 OR FB_MC2_AxisBasic_M_nMC_GearInMultiMaster_pMaster4 = 0 THEN
		M_nMC_GearInMultiMaster:= Tc3_HBI_System.cPOINTER_OR_INDEX_ERROR;
		RETURN;
	ELSE
		// AdvancedSlaveDynamics mode
		FB_MC2_AxisBasic_M_nMC_GearInMultiMaster_fbMC_GearInMultiMaster.Options.AdvancedSlaveDynamics:= FB_MC2_AxisBasic_M_nMC_GearInMultiMaster_bAdvancedSlaveDynamics;

		// Dynamic control Master/Slave
		IF NOT FB_MC2_AxisBasic_M_nMC_GearInMultiMaster_bAdvancedSlaveDynamics THEN
			FB_MC2_AxisBasic_M_nMC_GearInMultiMaster_fbMC_GearInMultiMaster.Acceleration:= ABS(FB_MC2_AxisBasic_M_nMC_GearInMultiMaster_pMaster1^.NcToPlc.SetAcc);
			FB_MC2_AxisBasic_M_nMC_GearInMultiMaster_fbMC_GearInMultiMaster.Deceleration:= 0.0;
			FB_MC2_AxisBasic_M_nMC_GearInMultiMaster_fbMC_GearInMultiMaster.Jerk:= ABS(FB_MC2_AxisBasic_M_nMC_GearInMultiMaster_pMaster1^.NcToPlc.SetJerk);
		ELSE
			FB_MC2_AxisBasic_M_nMC_GearInMultiMaster_fbMC_GearInMultiMaster.Acceleration:= _stDynamic.lrAcceleration;
			FB_MC2_AxisBasic_M_nMC_GearInMultiMaster_fbMC_GearInMultiMaster.Deceleration:= _stDynamic.lrDeceleration;
			FB_MC2_AxisBasic_M_nMC_GearInMultiMaster_fbMC_GearInMultiMaster.Jerk:= _stDynamic.lrJerk;
		END_IF
	
		// Reset
		IF _bReset THEN
			// Error
			IF FB_MC2_AxisBasic_M_nMC_GearInMultiMaster_fbMC_GearInMultiMaster.Error THEN
				FB_MC2_AxisBasic_M_nMC_GearInMultiMaster_fbMC_GearInMultiMaster(
					Master1:= FB_MC2_AxisBasic_M_nMC_GearInMultiMaster_pMaster1^,
					Master2:= FB_MC2_AxisBasic_M_nMC_GearInMultiMaster_pMaster2^, 
					Master3:= FB_MC2_AxisBasic_M_nMC_GearInMultiMaster_pMaster3^, 
					Master4:= FB_MC2_AxisBasic_M_nMC_GearInMultiMaster_pMaster4^, 
					Slave:= _stAXIS_REF, 
					Enable:= FALSE, 
					GearRatio1:= FB_MC2_AxisBasic_M_nMC_GearInMultiMaster_lrGearRatio1, 
					GearRatio2:= FB_MC2_AxisBasic_M_nMC_GearInMultiMaster_lrGearRatio2, 
					GearRatio3:= FB_MC2_AxisBasic_M_nMC_GearInMultiMaster_lrGearRatio3, 
					GearRatio4:= FB_MC2_AxisBasic_M_nMC_GearInMultiMaster_lrGearRatio4, 
					// Acceleration:= _stDynamic.lrAcceleration, 
					// Deceleration:= _stDynamic.lrDeceleration, 
					// Jerk:= _stDynamic.lrJerk, 
					BufferMode:= , 
					InGear=> , 
					Busy=> , 
					Active=> , 
					CommandAborted=> , 
					Error=> , 
					ErrorID=> );
			ELSE
				// Not Error
				FB_MC2_AxisBasic_M_nMC_GearInMultiMaster_fbMC_GearInMultiMaster(
					Master1:= FB_MC2_AxisBasic_M_nMC_GearInMultiMaster_pMaster1^,
					Master2:= FB_MC2_AxisBasic_M_nMC_GearInMultiMaster_pMaster2^, 
					Master3:= FB_MC2_AxisBasic_M_nMC_GearInMultiMaster_pMaster3^, 
					Master4:= FB_MC2_AxisBasic_M_nMC_GearInMultiMaster_pMaster4^, 
					Slave:= _stAXIS_REF, 
					Enable:= FB_MC2_AxisBasic_M_nMC_GearInMultiMaster_bEnable, 
					GearRatio1:= FB_MC2_AxisBasic_M_nMC_GearInMultiMaster_lrGearRatio1, 
					GearRatio2:= FB_MC2_AxisBasic_M_nMC_GearInMultiMaster_lrGearRatio2, 
					GearRatio3:= FB_MC2_AxisBasic_M_nMC_GearInMultiMaster_lrGearRatio3, 
					GearRatio4:= FB_MC2_AxisBasic_M_nMC_GearInMultiMaster_lrGearRatio4,
					// Acceleration:= _stDynamic.lrAcceleration, 
					// Deceleration:= _stDynamic.lrDeceleration, 
					// Jerk:= _stDynamic.lrJerk, 
					BufferMode:= , 
					InGear=> , 
					Busy=> , 
					Active=> , 
					CommandAborted=> , 
					Error=> , 
					ErrorID=> );
			END_IF
		ELSE
			// Gear in
			FB_MC2_AxisBasic_M_nMC_GearInMultiMaster_fbMC_GearInMultiMaster(
				Master1:= FB_MC2_AxisBasic_M_nMC_GearInMultiMaster_pMaster1^,
				Master2:= FB_MC2_AxisBasic_M_nMC_GearInMultiMaster_pMaster2^, 
				Master3:= FB_MC2_AxisBasic_M_nMC_GearInMultiMaster_pMaster3^, 
				Master4:= FB_MC2_AxisBasic_M_nMC_GearInMultiMaster_pMaster4^, 
				Slave:= _stAXIS_REF, 
				Enable:= FB_MC2_AxisBasic_M_nMC_GearInMultiMaster_bEnable, 
				GearRatio1:= FB_MC2_AxisBasic_M_nMC_GearInMultiMaster_lrGearRatio1, 
				GearRatio2:= FB_MC2_AxisBasic_M_nMC_GearInMultiMaster_lrGearRatio2, 
				GearRatio3:= FB_MC2_AxisBasic_M_nMC_GearInMultiMaster_lrGearRatio3, 
				GearRatio4:= FB_MC2_AxisBasic_M_nMC_GearInMultiMaster_lrGearRatio4,
				// Acceleration:= _stDynamic.lrAcceleration, 
				// Deceleration:= _stDynamic.lrDeceleration, 
				// Jerk:= _stDynamic.lrJerk, 
				BufferMode:= , 
				InGear=> , 
				Busy=> , 
				Active=> , 
				CommandAborted=> , 
				Error=> , 
				ErrorID=> );
		END_IF
		
		// Error	
		IF FB_MC2_AxisBasic_M_nMC_GearInMultiMaster_fbMC_GearInMultiMaster.Error THEN
			M_nError(nErrorID:= FB_MC2_AxisBasic_M_nMC_GearInMultiMaster_fbMC_GearInMultiMaster.ErrorID);
			M_nMC_GearInMultiMaster:= FB_MC2_AxisBasic_M_nMC_GearInMultiMaster_fbMC_GearInMultiMaster.ErrorID;
		ELSE
			// Done
			IF FB_MC2_AxisBasic_M_nMC_GearInMultiMaster_fbMC_GearInMultiMaster.CommandAborted THEN
				M_nMC_GearInMultiMaster:= Tc3_HBI_System.cABORTED;
			ELSE
				IF FB_MC2_AxisBasic_M_nMC_GearInMultiMaster_bEnable THEN
					IF _stAXIS_REF.Status.Coupled AND FB_MC2_AxisBasic_M_nMC_GearInMultiMaster_fbMC_GearInMultiMaster.InGear THEN
						M_nMC_GearInMultiMaster:= Tc3_HBI_System.cCOMPLETE;
					ELSE
						M_nMC_GearInMultiMaster:= Tc3_HBI_System.cRUNNING;
					END_IF
				ELSE
					M_nMC_GearInMultiMaster:= Tc3_HBI_System.cIDLE;
				END_IF
			END_IF
		END_IF	
		
	END_IF
ELSE	
	FB_MC2_AxisBasic_M_nMC_GearInMultiMaster_fbMC_GearInMultiMaster(Master1:= FB_MC2_AxisBasic_M_nMC_GearInMultiMaster_pMaster1^, Master2:= FB_MC2_AxisBasic_M_nMC_GearInMultiMaster_pMaster2^, Master3:= FB_MC2_AxisBasic_M_nMC_GearInMultiMaster_pMaster3^, Master4:= FB_MC2_AxisBasic_M_nMC_GearInMultiMaster_pMaster4^, Slave:= _stAXIS_REF, Enable:= FALSE);
	IF FB_MC2_AxisBasic_M_nMC_GearInMultiMaster_bEnable THEN
		M_nMC_GearInMultiMaster:= Tc3_HBI_System.cMAPPING_ERROR;
	END_IF
	RETURN;
END_IF
END_METHOD

//	The result of the method is an unsigned double integer
//	0 = idle 
//	1 = coupled
//	2 = starting
//	3 = running
//	4 = aborted
// 	5 = no hardware connected
// 	6 = Spare
//	7 = pointer or index error
//	8 = mapping error
//	9 = parameter error
//	10 = complete
//	Any other number = ErrorID
METHOD PUBLIC M_nMC_GearOut : UDINT
VAR_INPUT
	bExecute: BOOL;
END_VAR
// Local variable
FB_MC2_AxisBasic_M_nMC_GearOut_bExecute:= bExecute;

// Reset
IF _bReset THEN
	IF FB_MC2_AxisBasic_M_nMC_GearOut_fbMC2_GearOut.Error THEN
		// Gear out
		FB_MC2_AxisBasic_M_nMC_GearOut_fbMC2_GearOut(
			Slave:= _stAXIS_REF, 
			Execute:= FALSE, 
			Options:= , 
			Done=> , 
			Busy=> , 
			Error=> , 
			ErrorID=> );
	ELSE
		// Gear out
		IF _stAXIS_REF.NcToPlc.AxisID > 0 THEN
			FB_MC2_AxisBasic_M_nMC_GearOut_fbMC2_GearOut(
				Slave:= _stAXIS_REF, 
				Execute:= FB_MC2_AxisBasic_M_nMC_GearOut_bExecute, 
				Options:= , 
				Done=> , 
				Busy=> , 
				Error=> , 
				ErrorID=> );
		ELSE
			FB_MC2_AxisBasic_M_nMC_GearOut_fbMC2_GearOut(Slave:= _stAXIS_REF, Execute:= bExecute); 
			IF FB_MC2_AxisBasic_M_nMC_GearOut_bExecute THEN
				M_nMC_GearOut:= Tc3_HBI_System.cMAPPING_ERROR;
			END_IF
			RETURN;
		END_IF
	END_IF	
ELSE
	// Gear out
	IF _stAXIS_REF.NcToPlc.AxisID > 0 THEN
		FB_MC2_AxisBasic_M_nMC_GearOut_fbMC2_GearOut(
			Slave:= _stAXIS_REF, 
			Execute:= FB_MC2_AxisBasic_M_nMC_GearOut_bExecute, 
			Options:= , 
			Done=> , 
			Busy=> , 
			Error=> , 
			ErrorID=> );
	ELSE
		FB_MC2_AxisBasic_M_nMC_GearOut_fbMC2_GearOut(Slave:= _stAXIS_REF, Execute:= FB_MC2_AxisBasic_M_nMC_GearOut_bExecute); 
		IF FB_MC2_AxisBasic_M_nMC_GearOut_bExecute THEN
			M_nMC_GearOut:= Tc3_HBI_System.cMAPPING_ERROR;
		END_IF
		RETURN;
	END_IF
END_IF

// Error	
IF FB_MC2_AxisBasic_M_nMC_GearOut_fbMC2_GearOut.Error THEN
	M_nError(nErrorID:= FB_MC2_AxisBasic_M_nMC_GearOut_fbMC2_GearOut.ErrorID);
	M_nMC_GearOut:= FB_MC2_AxisBasic_M_nMC_GearOut_fbMC2_GearOut.ErrorID;
ELSE
	// Done
	IF FB_MC2_AxisBasic_M_nMC_GearOut_bExecute THEN
		IF FB_MC2_AxisBasic_M_nMC_GearOut_fbMC2_GearOut.Done AND NOT _stAXIS_REF.Status.Coupled THEN
			M_nMC_GearOut:= Tc3_HBI_System.cCOMPLETE;
		ELSE
			M_nMC_GearOut:= Tc3_HBI_System.cRUNNING;
		END_IF
	END_IF
END_IF
END_METHOD

//	The result of the method is an unsigned double integer
//	0 = idle 
//	1 = coupled
//	2 = starting
//	3 = running
//	4 = aborted
// 	5 = no hardware connected
// 	6 = Spare
//	7 = pointer or index error
//	8 = mapping error
//	9 = parameter error
//	10 = complete
//	Any other number = ErrorID
METHOD PUBLIC M_nMC_InverseMotor : UDINT
VAR_INPUT
	bExecute: BOOL;
	bInverse: BOOL;
END_VAR
// Local variable
FB_MC2_AxisBasic_M_nMC_InverseMotor_bExecute:= bExecute;
FB_MC2_AxisBasic_M_nMC_InverseMotor_bInverse:= bInverse;

//**********************************
// Reset 
//**********************************
IF _bReset THEN
	IF _bError THEN	
		FB_MC2_AxisBasic_M_nMC_InverseMotor_fbADSRDWRT(WRTRD:= FALSE);
		FB_MC2_AxisBasic_M_nMC_InverseMotor_iState:= 000;
	END_IF
END_IF

//**********************************
// Wait for execute
//**********************************
IF _stAXIS_REF.NcToPlc.AxisID > 0 THEN
	FB_MC2_AxisBasic_M_nMC_InverseMotor_fbExecute_R_TRIG(CLK:= FB_MC2_AxisBasic_M_nMC_InverseMotor_bExecute);
	IF FB_MC2_AxisBasic_M_nMC_InverseMotor_fbExecute_R_TRIG.Q THEN
		FB_MC2_AxisBasic_M_nMC_InverseMotor_fbADSRDWRT(WRTRD:= FALSE); 
		
		// Axis not coupled	
		IF NOT _stAXIS_REF.Status.Coupled THEN
			FB_MC2_AxisBasic_M_nMC_InverseMotor_iState:= 001;
		ELSE
			FB_MC2_AxisBasic_M_nMC_InverseMotor_iState:= 010;
		END_IF
	
	END_IF
ELSE
	FB_MC2_AxisBasic_M_nMC_InverseMotor_fbExecute_R_TRIG(CLK:= FALSE);
	FB_MC2_AxisBasic_M_nMC_InverseMotor_iState:= 000;
	IF FB_MC2_AxisBasic_M_nMC_InverseMotor_bExecute THEN
		M_nMC_InverseMotor:= Tc3_HBI_System.cMAPPING_ERROR;
	END_IF
	RETURN;
END_IF


//**********************************
// Main sequence
//**********************************
CASE FB_MC2_AxisBasic_M_nMC_InverseMotor_iState OF

	000: 	// Do nothing
	
	001:	// Parameter setup
			M_nMC_InverseMotor:= Tc3_HBI_System.cRUNNING;
			IF _stAXIS_REF.NcToPlc.AxisID > 0 THEN
				(* Copy values to transfer *)
				FB_MC2_AxisBasic_M_nMC_InverseMotor_stMC2_Param.nEncoderDir:= BOOL_TO_WORD(FB_MC2_AxisBasic_M_nMC_InverseMotor_bInverse);
				FB_MC2_AxisBasic_M_nMC_InverseMotor_stMC2_Param.nMotorDir:= BOOL_TO_WORD(FB_MC2_AxisBasic_M_nMC_InverseMotor_bInverse);
				FB_MC2_AxisBasic_M_nMC_InverseMotor_stMC2_Param.nHomeCamDir:= BOOL_TO_WORD( FB_MC2_AxisBasic_M_nMC_InverseMotor_bInverse);
				FB_MC2_AxisBasic_M_nMC_InverseMotor_stMC2_Param.nHomeSyncDir:= BOOL_TO_WORD(NOT FB_MC2_AxisBasic_M_nMC_InverseMotor_bInverse);
			
				// Setup adresses for transfer - The lines must be in the same order as the struct
				_iIdx:= 1;
				FB_MC2_AxisBasic_M_nMC_InverseMotor_stMC2_Param.aParm[_iIdx].nIndexGroup:= 16#00005000 + _stAXIS_REF.NcToPlc.AxisId; 	FB_MC2_AxisBasic_M_nMC_InverseMotor_stMC2_Param.aParm[_iIdx].nIndexOffset:= 16#00000008;	FB_MC2_AxisBasic_M_nMC_InverseMotor_stMC2_Param.aParm[_iIdx].nDataSize:= SIZEOF(FB_MC2_AxisBasic_M_nMC_InverseMotor_stMC2_Param.nEncoderDir);	_iIdx := _iIdx+1;
				FB_MC2_AxisBasic_M_nMC_InverseMotor_stMC2_Param.aParm[_iIdx].nIndexGroup:= 16#00007000 + _stAXIS_REF.NcToPlc.AxisId; 	FB_MC2_AxisBasic_M_nMC_InverseMotor_stMC2_Param.aParm[_iIdx].nIndexOffset:= 16#00000006;	FB_MC2_AxisBasic_M_nMC_InverseMotor_stMC2_Param.aParm[_iIdx].nDataSize:= SIZEOF(FB_MC2_AxisBasic_M_nMC_InverseMotor_stMC2_Param.nMotorDir);		_iIdx := _iIdx+1;
				FB_MC2_AxisBasic_M_nMC_InverseMotor_stMC2_Param.aParm[_iIdx].nIndexGroup:= 16#00005000 + _stAXIS_REF.NcToPlc.AxisId; 	FB_MC2_AxisBasic_M_nMC_InverseMotor_stMC2_Param.aParm[_iIdx].nIndexOffset:= 16#00000101;	FB_MC2_AxisBasic_M_nMC_InverseMotor_stMC2_Param.aParm[_iIdx].nDataSize:= SIZEOF(FB_MC2_AxisBasic_M_nMC_InverseMotor_stMC2_Param.nHomeCamDir);	_iIdx := _iIdx+1;
				FB_MC2_AxisBasic_M_nMC_InverseMotor_stMC2_Param.aParm[_iIdx].nIndexGroup:= 16#00005000 + _stAXIS_REF.NcToPlc.AxisId; 	FB_MC2_AxisBasic_M_nMC_InverseMotor_stMC2_Param.aParm[_iIdx].nIndexOffset:= 16#00000102;	FB_MC2_AxisBasic_M_nMC_InverseMotor_stMC2_Param.aParm[_iIdx].nDataSize:= SIZEOF(FB_MC2_AxisBasic_M_nMC_InverseMotor_stMC2_Param.nHomeSyncDir);	_iIdx := _iIdx+1;
		
				FB_MC2_AxisBasic_M_nMC_InverseMotor_iState:= 002;
			END_IF
	
	002:	// Write ADS list 
			M_nMC_InverseMotor:= Tc3_HBI_System.cRUNNING;
			FB_MC2_AxisBasic_M_nMC_InverseMotor_fbADSRDWRT(WRTRD:= FALSE);
			FB_MC2_AxisBasic_M_nMC_InverseMotor_fbADSRDWRT(
				NETID:= '', 
				PORT:= 501,
				IDXGRP:= 16#F081, 	// Write list 
				IDXOFFS:= SIZEOF(FB_MC2_AxisBasic_M_nMC_InverseMotor_arr_nADSReturn) / SIZEOF(FB_MC2_AxisBasic_M_nMC_InverseMotor_arr_nADSReturn[1]),
				WRITELEN:= SIZEOF(FB_MC2_AxisBasic_M_nMC_InverseMotor_stMC2_Param),
				READLEN:= SIZEOF(FB_MC2_AxisBasic_M_nMC_InverseMotor_arr_nADSReturn),
				SRCADDR:= ADR(FB_MC2_AxisBasic_M_nMC_InverseMotor_stMC2_Param),
				DESTADDR:= ADR(FB_MC2_AxisBasic_M_nMC_InverseMotor_arr_nADSReturn),
				WRTRD:= TRUE, 
				TMOUT:= T#2S); 
	
			FB_MC2_AxisBasic_M_nMC_InverseMotor_iState:= 003;

	003:	// Done		
			M_nMC_InverseMotor:= Tc3_HBI_System.cRUNNING;
			FB_MC2_AxisBasic_M_nMC_InverseMotor_fbADSRDWRT(WRTRD:= TRUE);
	
			// Error handling
			IF FB_MC2_AxisBasic_M_nMC_InverseMotor_fbADSRDWRT.ERR THEN
				M_nError(nErrorID:= FB_MC2_AxisBasic_M_nMC_InverseMotor_fbADSRDWRT.ERRID);
				M_nMC_InverseMotor:= FB_MC2_AxisBasic_M_nMC_InverseMotor_fbADSRDWRT.ERRID;
			ELSE
				// Done
				IF NOT FB_MC2_AxisBasic_M_nMC_InverseMotor_fbADSRDWRT.BUSY THEN
					FB_MC2_AxisBasic_M_nMC_InverseMotor_fbADSRDWRT(WRTRD:= FALSE);
					FB_MC2_AxisBasic_M_nMC_InverseMotor_iState:= 004;
				END_IF
			END_IF
	
	004:	// Write list error handling
			M_nMC_InverseMotor:= Tc3_HBI_System.cRUNNING;
			FOR _iIdx := 1 TO UDINT_TO_INT(FB_MC2_AxisBasic_M_nMC_InverseMotor_fbADSRDWRT.IDXOFFS) DO
				IF FB_MC2_AxisBasic_M_nMC_InverseMotor_arr_nADSReturn[_iIdx] > 16#00 THEN
					M_nError(nErrorID:= FB_MC2_AxisBasic_M_nMC_InverseMotor_arr_nADSReturn[_iIdx]);
				END_IF
			END_FOR	
			FB_MC2_AxisBasic_M_nMC_InverseMotor_iState:= 005;
		
	005:	// Write list error handling	
			M_nMC_InverseMotor:= Tc3_HBI_System.cRUNNING;
			IF NOT _bError THEN
				FB_MC2_AxisBasic_M_nMC_InverseMotor_iState:= 020;
			ELSE
				M_nMC_InverseMotor:= _nErrorID;
				IF NOT FB_MC2_AxisBasic_M_nMC_InverseMotor_bExecute THEN
					FB_MC2_AxisBasic_M_nMC_InverseMotor_iState:= 000;
				END_IF
			END_IF
		
	010:	// Coupled
			M_nMC_InverseMotor:= Tc3_HBI_System.cCOUPLED;
			IF NOT FB_MC2_AxisBasic_M_nMC_InverseMotor_bExecute THEN
				FB_MC2_AxisBasic_M_nMC_InverseMotor_fbADSRDWRT(WRTRD:= FALSE); 
				FB_MC2_AxisBasic_M_nMC_InverseMotor_iState:= 000;
			END_IF	

	020:	// Done
			M_nMC_InverseMotor:= Tc3_HBI_System.cCOMPLETE;
			
			IF NOT FB_MC2_AxisBasic_M_nMC_InverseMotor_bExecute THEN
				FB_MC2_AxisBasic_M_nMC_InverseMotor_fbADSRDWRT(WRTRD:= FALSE); 
				FB_MC2_AxisBasic_M_nMC_InverseMotor_iState:= 000;
			END_IF	
		
ELSE
	FB_MC2_AxisBasic_M_nMC_InverseMotor_iState:= 000;
END_CASE
END_METHOD

//	The result of the method is an unsigned double integer
//	0 = idle 
//	1 = coupled
//	2 = starting
//	3 = running
//	4 = aborted
// 	5 = no hardware connected
// 	6 = Spare
//	7 = pointer or index error
//	8 = mapping error
//	9 = parameter error
//	10 = complete
//	Any other number = ErrorID
METHOD PUBLIC M_nMC_PhasingAbsolute : UDINT
VAR_INPUT
	bExecute: BOOL;
	pMaster: POINTER TO TC2_MC2.AXIS_REF;
	lrPhaseShift: LREAL;
	lrVelocity: LREAL;
END_VAR
// Local variable
FB_MC2_AxisBasic_M_nMC_PhasingAbsolute_bExecute:= bExecute;
FB_MC2_AxisBasic_M_nMC_PhasingAbsolute_pMaster:= pMaster;
FB_MC2_AxisBasic_M_nMC_PhasingAbsolute_lrPhaseShift:= lrPhaseShift;
FB_MC2_AxisBasic_M_nMC_PhasingAbsolute_lrVelocity:= lrVelocity;

//**********************************
// Axis check
//**********************************
IF _stAXIS_REF.NcToPlc.AxisID = 0 THEN
	M_nMC_PhasingAbsolute:= Tc3_HBI_System.cMAPPING_ERROR;
	FB_MC2_AxisBasic_M_nMC_PhasingAbsolute_iState:= 000;
	RETURN;		
END_IF

//**********************************
// Pointer check
//**********************************
IF FB_MC2_AxisBasic_M_nMC_PhasingAbsolute_pMaster = 0 THEN
	M_nMC_PhasingAbsolute:= Tc3_HBI_System.cPOINTER_OR_INDEX_ERROR;
	FB_MC2_AxisBasic_M_nMC_PhasingAbsolute_iState:= 000;
	RETURN;
END_IF

//**********************************
// Reset 
//**********************************
IF _bReset THEN
	IF _bError THEN
		FB_MC2_AxisBasic_M_nMC_PhasingAbsolute_fbMC2_HaltParsing(Master:= FB_MC2_AxisBasic_M_nMC_PhasingAbsolute_pMaster^, Slave:= _stAXIS_REF, Execute:= FALSE); 
		FB_MC2_AxisBasic_M_nMC_PhasingAbsolute_fbMC2_PhasingAbsolute(Master:= FB_MC2_AxisBasic_M_nMC_PhasingAbsolute_pMaster^, Slave:= _stAXIS_REF, Execute:= FALSE); 
		FB_MC2_AxisBasic_M_nMC_PhasingAbsolute_iState:= 000;
	END_IF
END_IF

//**********************************
// Wait for execute
//**********************************
IF _stAXIS_REF.NcToPlc.AxisID > 0 THEN
	FB_MC2_AxisBasic_M_nMC_PhasingAbsolute_fbExecute_R_TRIG(CLK:= FB_MC2_AxisBasic_M_nMC_PhasingAbsolute_bExecute);
	IF FB_MC2_AxisBasic_M_nMC_PhasingAbsolute_fbExecute_R_TRIG.Q THEN
		FB_MC2_AxisBasic_M_nMC_PhasingAbsolute_fbMC2_HaltParsing(Master:= FB_MC2_AxisBasic_M_nMC_PhasingAbsolute_pMaster^, Slave:= _stAXIS_REF, Execute:= FALSE); 
		FB_MC2_AxisBasic_M_nMC_PhasingAbsolute_fbMC2_PhasingAbsolute(Master:= FB_MC2_AxisBasic_M_nMC_PhasingAbsolute_pMaster^, Slave:= _stAXIS_REF, Execute:= FALSE); 
		FB_MC2_AxisBasic_M_nMC_PhasingAbsolute_iState:= 010;
	END_IF
	FB_MC2_AxisBasic_M_nMC_PhasingAbsolute_fbNotExecute_R_TRIG(CLK:= NOT FB_MC2_AxisBasic_M_nMC_PhasingAbsolute_bExecute);
	IF FB_MC2_AxisBasic_M_nMC_PhasingAbsolute_fbNotExecute_R_TRIG.Q THEN
		FB_MC2_AxisBasic_M_nMC_PhasingAbsolute_fbMC2_HaltParsing(Master:= FB_MC2_AxisBasic_M_nMC_PhasingAbsolute_pMaster^, Slave:= _stAXIS_REF, Execute:= FALSE); 
		FB_MC2_AxisBasic_M_nMC_PhasingAbsolute_fbMC2_PhasingAbsolute(Master:= FB_MC2_AxisBasic_M_nMC_PhasingAbsolute_pMaster^, Slave:= _stAXIS_REF, Execute:= FALSE); 
		FB_MC2_AxisBasic_M_nMC_PhasingAbsolute_lrAbsolutePhaseShift:= 0.0;
		IF FB_MC2_AxisBasic_M_nMC_PhasingAbsolute_fbMC2_PhasingAbsolute.Busy THEN
			FB_MC2_AxisBasic_M_nMC_PhasingAbsolute_iState:= 001;
		ELSE
			FB_MC2_AxisBasic_M_nMC_PhasingAbsolute_iState:= 000;
		END_IF
	END_IF
ELSE
	FB_MC2_AxisBasic_M_nMC_PhasingAbsolute_fbMC2_HaltParsing(Master:= FB_MC2_AxisBasic_M_nMC_PhasingAbsolute_pMaster^, Slave:= _stAXIS_REF, Execute:= FALSE); 
	FB_MC2_AxisBasic_M_nMC_PhasingAbsolute_fbMC2_PhasingAbsolute(Master:= FB_MC2_AxisBasic_M_nMC_PhasingAbsolute_pMaster^, Slave:= _stAXIS_REF, Execute:= FALSE); 
	FB_MC2_AxisBasic_M_nMC_PhasingAbsolute_lrAbsolutePhaseShift:= 0.0;
	FB_MC2_AxisBasic_M_nMC_PhasingAbsolute_iState:= 000;
	IF FB_MC2_AxisBasic_M_nMC_PhasingAbsolute_bExecute THEN
		M_nMC_PhasingAbsolute:= Tc3_HBI_System.cMAPPING_ERROR;
	END_IF
	RETURN;
END_IF


//**********************************
// Main sequence
//**********************************
CASE FB_MC2_AxisBasic_M_nMC_PhasingAbsolute_iState OF

	000: 	// Do nothing
	
	001:	// Abort ParshingRelative
			M_nMC_PhasingAbsolute:= Tc3_HBI_System.cSTARTING;
			IF _stAXIS_REF.Status.Coupled THEN
				FB_MC2_AxisBasic_M_nMC_PhasingAbsolute_fbMC2_HaltParsing(Master:= FB_MC2_AxisBasic_M_nMC_PhasingAbsolute_pMaster^, Slave:= _stAXIS_REF, Execute:= FALSE);
				FB_MC2_AxisBasic_M_nMC_PhasingAbsolute_fbMC2_HaltParsing(
					Master:= FB_MC2_AxisBasic_M_nMC_PhasingAbsolute_pMaster^, 
					Slave:= _stAXIS_REF, 
					Execute:= TRUE, 
					Deceleration:= _stDynamic.lrDeceleration, 
					Jerk:= _stDynamic.lrJerk, 
					BufferMode:= , 
					Options:= , 
					Done=> , 
					Busy=> , 
					Active=> , 
					CommandAborted=> , 
					Error=> , 
					ErrorID=> );
					
				FB_MC2_AxisBasic_M_nMC_PhasingAbsolute_iState:= FB_MC2_AxisBasic_M_nMC_PhasingAbsolute_iState +1;
			ELSE
				FB_MC2_AxisBasic_M_nMC_PhasingAbsolute_iState:= 000;	
			END_IF
			
	002:	// Abort ParshingAbsolute - Done
			M_nMC_PhasingAbsolute:= Tc3_HBI_System.cRUNNING;
			FB_MC2_AxisBasic_M_nMC_PhasingAbsolute_fbMC2_HaltParsing(Master:= FB_MC2_AxisBasic_M_nMC_PhasingAbsolute_pMaster^, Slave:= _stAXIS_REF, Execute:= TRUE);

			// Error handling
			IF FB_MC2_AxisBasic_M_nMC_PhasingAbsolute_fbMC2_HaltParsing.Error THEN
				M_nError(nErrorID:= FB_MC2_AxisBasic_M_nMC_PhasingAbsolute_fbMC2_HaltParsing.ErrorID);
				M_nMC_PhasingAbsolute:= FB_MC2_AxisBasic_M_nMC_PhasingAbsolute_fbMC2_HaltParsing.ErrorID;
			ELSE
				// Done
				IF FB_MC2_AxisBasic_M_nMC_PhasingAbsolute_fbMC2_HaltParsing.Done THEN
					FB_MC2_AxisBasic_M_nMC_PhasingAbsolute_fbMC2_HaltParsing(Master:= FB_MC2_AxisBasic_M_nMC_PhasingAbsolute_pMaster^, Slave:= _stAXIS_REF, Execute:= FALSE);
					FB_MC2_AxisBasic_M_nMC_PhasingAbsolute_iState:= 000;	
				END_IF
			END_IF
			
	010:	// ParshingAbsolute
			M_nMC_PhasingAbsolute:= Tc3_HBI_System.cSTARTING;
			FB_MC2_AxisBasic_M_nMC_PhasingAbsolute_fbMC2_PhasingAbsolute(Master:= FB_MC2_AxisBasic_M_nMC_PhasingAbsolute_pMaster^, Slave:= _stAXIS_REF, Execute:= FALSE); 
			FB_MC2_AxisBasic_M_nMC_PhasingAbsolute_fbMC2_PhasingAbsolute(
				Master:= FB_MC2_AxisBasic_M_nMC_PhasingAbsolute_pMaster^, 
				Slave:= _stAXIS_REF, 
				Execute:= TRUE, 
				PhaseShift:= FB_MC2_AxisBasic_M_nMC_PhasingAbsolute_lrPhaseShift, 
				Velocity:= FB_MC2_AxisBasic_M_nMC_PhasingAbsolute_lrVelocity, 
				Acceleration:= _stDynamic.lrAcceleration, 
				Deceleration:= _stDynamic.lrDeceleration, 
				Jerk:= _stDynamic.lrJerk, 
				BufferMode:= , 
				Options:= , 
				Done=> , 
				Busy=> , 
				Active=> , 
				CommandAborted=> , 
				Error=> , 
				ErrorID=> , 
				AbsolutePhaseShift=> );

			FB_MC2_AxisBasic_M_nMC_PhasingAbsolute_iState:= FB_MC2_AxisBasic_M_nMC_PhasingAbsolute_iState +1;
	
	011:	// ParshingAbsolute - Done
			M_nMC_PhasingAbsolute:= Tc3_HBI_System.cRUNNING;
			FB_MC2_AxisBasic_M_nMC_PhasingAbsolute_fbMC2_PhasingAbsolute(Master:= FB_MC2_AxisBasic_M_nMC_PhasingAbsolute_pMaster^, Slave:= _stAXIS_REF, Execute:= TRUE, AbsolutePhaseShift=> FB_MC2_AxisBasic_M_nMC_PhasingAbsolute_lrAbsolutePhaseShift); 
	
			// Command aborted
			IF FB_MC2_AxisBasic_M_nMC_PhasingAbsolute_fbMC2_PhasingAbsolute.CommandAborted THEN
				FB_MC2_AxisBasic_M_nMC_PhasingAbsolute_iState:= 030;
			ELSE
				// Error handling
				IF FB_MC2_AxisBasic_M_nMC_PhasingAbsolute_fbMC2_PhasingAbsolute.Error THEN
					M_nError(nErrorID:= FB_MC2_AxisBasic_M_nMC_PhasingAbsolute_fbMC2_PhasingAbsolute.ErrorID);
					M_nMC_PhasingAbsolute:= FB_MC2_AxisBasic_M_nMC_PhasingAbsolute_fbMC2_PhasingAbsolute.ErrorID;
				ELSE
					// Done
					IF FB_MC2_AxisBasic_M_nMC_PhasingAbsolute_fbMC2_PhasingAbsolute.Done THEN
						FB_MC2_AxisBasic_M_nMC_PhasingAbsolute_iState:= 030;
					END_IF
				END_IF
			END_IF

	030:	// Done
			M_nMC_PhasingAbsolute:= Tc3_HBI_System.cCOMPLETE;
			
			IF FB_MC2_AxisBasic_M_nMC_PhasingAbsolute_bExecute THEN
				IF FB_MC2_AxisBasic_M_nMC_PhasingAbsolute_fbMC2_PhasingAbsolute.CommandAborted THEN
					M_nMC_PhasingAbsolute:= Tc3_HBI_System.cABORTED;
				END_IF
			ELSE
				FB_MC2_AxisBasic_M_nMC_PhasingAbsolute_fbMC2_HaltParsing(Master:= FB_MC2_AxisBasic_M_nMC_PhasingAbsolute_pMaster^, Slave:= _stAXIS_REF, Execute:= FALSE); 
				FB_MC2_AxisBasic_M_nMC_PhasingAbsolute_fbMC2_PhasingAbsolute(Master:= FB_MC2_AxisBasic_M_nMC_PhasingAbsolute_pMaster^, Slave:= _stAXIS_REF, Execute:= FALSE); 
				FB_MC2_AxisBasic_M_nMC_PhasingAbsolute_iState:= 000;
			END_IF	

ELSE
	FB_MC2_AxisBasic_M_nMC_PhasingAbsolute_iState:= 000;
END_CASE
END_METHOD

//	The result of the method is an unsigned double integer
//	0 = idle 
//	1 = coupled
//	2 = starting
//	3 = running
//	4 = aborted
// 	5 = no hardware connected
// 	6 = Spare
//	7 = pointer or index error
//	8 = mapping error
//	9 = parameter error
//	10 = complete
//	Any other number = ErrorID
METHOD PUBLIC M_nMC_PhasingRelative : UDINT
VAR_INPUT
	bExecute: BOOL;
	pMaster: POINTER TO TC2_MC2.AXIS_REF;
	lrPhaseShift: LREAL;
	lrVelocity: LREAL;
END_VAR
// Local variable
FB_MC2_AxisBasic_M_nMC_PhasingRelative_bExecute:= bExecute;
FB_MC2_AxisBasic_M_nMC_PhasingRelative_pMaster:= pMaster;
FB_MC2_AxisBasic_M_nMC_PhasingRelative_lrPhaseShift:= lrPhaseShift;
FB_MC2_AxisBasic_M_nMC_PhasingRelative_lrVelocity:= lrVelocity;

//**********************************
// Axis check
//**********************************
IF _stAXIS_REF.NcToPlc.AxisID = 0 THEN
	M_nMC_PhasingRelative:= Tc3_HBI_System.cMAPPING_ERROR;
	FB_MC2_AxisBasic_M_nMC_PhasingRelative_iState:= 000;
	RETURN;		
END_IF

//**********************************
// Pointer check
//**********************************
IF FB_MC2_AxisBasic_M_nMC_PhasingRelative_pMaster = 0 THEN
	M_nMC_PhasingRelative:= Tc3_HBI_System.cPOINTER_OR_INDEX_ERROR;
	FB_MC2_AxisBasic_M_nMC_PhasingRelative_iState:= 000;
	RETURN;
END_IF

//**********************************
// Reset 
//**********************************
IF _bReset THEN
	IF _bError THEN
		FB_MC2_AxisBasic_M_nMC_PhasingRelative_fbMC2_HaltParsing(Master:= FB_MC2_AxisBasic_M_nMC_PhasingRelative_pMaster^, Slave:= _stAXIS_REF, Execute:= FALSE); 
		FB_MC2_AxisBasic_M_nMC_PhasingRelative_fbMC2_PhasingRelative(Master:= FB_MC2_AxisBasic_M_nMC_PhasingRelative_pMaster^, Slave:= _stAXIS_REF, Execute:= FALSE); 
		FB_MC2_AxisBasic_M_nMC_PhasingRelative_iState:= 000;
	END_IF
END_IF

//**********************************
// Wait for execute
//**********************************
IF _stAXIS_REF.NcToPlc.AxisID > 0 THEN
	FB_MC2_AxisBasic_M_nMC_PhasingRelative_fbExecute_R_TRIG(CLK:= FB_MC2_AxisBasic_M_nMC_PhasingRelative_bExecute);
	IF FB_MC2_AxisBasic_M_nMC_PhasingRelative_fbExecute_R_TRIG.Q THEN
		FB_MC2_AxisBasic_M_nMC_PhasingRelative_fbMC2_HaltParsing(Master:= FB_MC2_AxisBasic_M_nMC_PhasingRelative_pMaster^, Slave:= _stAXIS_REF, Execute:= FALSE); 
		FB_MC2_AxisBasic_M_nMC_PhasingRelative_fbMC2_PhasingRelative(Master:= FB_MC2_AxisBasic_M_nMC_PhasingRelative_pMaster^, Slave:= _stAXIS_REF, Execute:= FALSE); 
		FB_MC2_AxisBasic_M_nMC_PhasingRelative_iState:= 010;
	END_IF
	FB_MC2_AxisBasic_M_nMC_PhasingRelative_fbNotExecute_R_TRIG(CLK:= NOT FB_MC2_AxisBasic_M_nMC_PhasingRelative_bExecute);
	IF FB_MC2_AxisBasic_M_nMC_PhasingRelative_fbNotExecute_R_TRIG.Q THEN
		FB_MC2_AxisBasic_M_nMC_PhasingRelative_fbMC2_HaltParsing(Master:= FB_MC2_AxisBasic_M_nMC_PhasingRelative_pMaster^, Slave:= _stAXIS_REF, Execute:= FALSE); 
		FB_MC2_AxisBasic_M_nMC_PhasingRelative_fbMC2_PhasingRelative(Master:= FB_MC2_AxisBasic_M_nMC_PhasingRelative_pMaster^, Slave:= _stAXIS_REF, Execute:= FALSE); 
		FB_MC2_AxisBasic_M_nMC_PhasingRelative_lrCoveredPhaseShift:= 0.0;
		IF FB_MC2_AxisBasic_M_nMC_PhasingRelative_fbMC2_PhasingRelative.Busy THEN
			FB_MC2_AxisBasic_M_nMC_PhasingRelative_iState:= 001;
		ELSE
			FB_MC2_AxisBasic_M_nMC_PhasingRelative_iState:= 000;
		END_IF
	END_IF
ELSE
	FB_MC2_AxisBasic_M_nMC_PhasingRelative_fbMC2_HaltParsing(Master:= FB_MC2_AxisBasic_M_nMC_PhasingRelative_pMaster^, Slave:= _stAXIS_REF, Execute:= FALSE); 
	FB_MC2_AxisBasic_M_nMC_PhasingRelative_fbMC2_PhasingRelative(Master:= FB_MC2_AxisBasic_M_nMC_PhasingRelative_pMaster^, Slave:= _stAXIS_REF, Execute:= FALSE); 
	FB_MC2_AxisBasic_M_nMC_PhasingRelative_lrCoveredPhaseShift:= 0.0;
	FB_MC2_AxisBasic_M_nMC_PhasingRelative_iState:= 000;
	IF FB_MC2_AxisBasic_M_nMC_PhasingRelative_bExecute THEN
		M_nMC_PhasingRelative:= Tc3_HBI_System.cMAPPING_ERROR;
	END_IF
	RETURN;
END_IF


//**********************************
// Main sequence
//**********************************
CASE FB_MC2_AxisBasic_M_nMC_PhasingRelative_iState OF

	000: 	// Do nothing
	
	001:	// Abort ParshingRelative
			M_nMC_PhasingRelative:= Tc3_HBI_System.cSTARTING;
			IF _stAXIS_REF.Status.Coupled THEN
				FB_MC2_AxisBasic_M_nMC_PhasingRelative_fbMC2_HaltParsing(Master:= FB_MC2_AxisBasic_M_nMC_PhasingRelative_pMaster^, Slave:= _stAXIS_REF, Execute:= FALSE);
				FB_MC2_AxisBasic_M_nMC_PhasingRelative_fbMC2_HaltParsing(
					Master:= FB_MC2_AxisBasic_M_nMC_PhasingRelative_pMaster^, 
					Slave:= _stAXIS_REF, 
					Execute:= TRUE, 
					Deceleration:= _stDynamic.lrDeceleration, 
					Jerk:= _stDynamic.lrJerk, 
					BufferMode:= , 
					Options:= , 
					Done=> , 
					Busy=> , 
					Active=> , 
					CommandAborted=> , 
					Error=> , 
					ErrorID=> );
					
				FB_MC2_AxisBasic_M_nMC_PhasingRelative_iState:= FB_MC2_AxisBasic_M_nMC_PhasingRelative_iState +1;
			ELSE
				FB_MC2_AxisBasic_M_nMC_PhasingRelative_iState:= 000;	
			END_IF			
			
	002:	// Abort ParshingRelative - Done
			M_nMC_PhasingRelative:= Tc3_HBI_System.cRUNNING;
			FB_MC2_AxisBasic_M_nMC_PhasingRelative_fbMC2_HaltParsing(Master:= FB_MC2_AxisBasic_M_nMC_PhasingRelative_pMaster^, Slave:= _stAXIS_REF, Execute:= TRUE);

			// Error handling
			IF FB_MC2_AxisBasic_M_nMC_PhasingRelative_fbMC2_HaltParsing.Error THEN
				M_nError(nErrorID:= FB_MC2_AxisBasic_M_nMC_PhasingRelative_fbMC2_HaltParsing.ErrorID);
				M_nMC_PhasingRelative:= FB_MC2_AxisBasic_M_nMC_PhasingRelative_fbMC2_HaltParsing.ErrorID;
			ELSE
				// Done
				IF FB_MC2_AxisBasic_M_nMC_PhasingRelative_fbMC2_HaltParsing.Done THEN
					FB_MC2_AxisBasic_M_nMC_PhasingRelative_fbMC2_HaltParsing(Master:= FB_MC2_AxisBasic_M_nMC_PhasingRelative_pMaster^, Slave:= _stAXIS_REF, Execute:= FALSE);
					FB_MC2_AxisBasic_M_nMC_PhasingRelative_iState:= 000;	
				END_IF
			END_IF
			
	010:	// ParshingRelative
			M_nMC_PhasingRelative:= Tc3_HBI_System.cSTARTING;
			FB_MC2_AxisBasic_M_nMC_PhasingRelative_fbMC2_PhasingRelative(Master:= FB_MC2_AxisBasic_M_nMC_PhasingRelative_pMaster^, Slave:= _stAXIS_REF, Execute:= FALSE); 
			FB_MC2_AxisBasic_M_nMC_PhasingRelative_fbMC2_PhasingRelative(
				Master:= FB_MC2_AxisBasic_M_nMC_PhasingRelative_pMaster^, 
				Slave:= _stAXIS_REF, 
				Execute:= TRUE, 
				PhaseShift:= FB_MC2_AxisBasic_M_nMC_PhasingRelative_lrPhaseShift, 
				Velocity:= FB_MC2_AxisBasic_M_nMC_PhasingRelative_lrVelocity, 
				Acceleration:= _stDynamic.lrAcceleration, 
				Deceleration:= _stDynamic.lrDeceleration, 
				Jerk:= _stDynamic.lrJerk, 
				BufferMode:= , 
				Options:= , 
				Done=> , 
				Busy=> , 
				Active=> , 
				CommandAborted=> , 
				Error=> , 
				ErrorID=> , 
				CoveredPhaseShift=> );

			FB_MC2_AxisBasic_M_nMC_PhasingRelative_iState:= FB_MC2_AxisBasic_M_nMC_PhasingRelative_iState +1;
	
	011:	// ParshingRelative - Done
			M_nMC_PhasingRelative:= Tc3_HBI_System.cRUNNING;
			FB_MC2_AxisBasic_M_nMC_PhasingRelative_fbMC2_PhasingRelative(Master:= FB_MC2_AxisBasic_M_nMC_PhasingRelative_pMaster^, Slave:= _stAXIS_REF, Execute:= TRUE, CoveredPhaseShift=> FB_MC2_AxisBasic_M_nMC_PhasingRelative_lrCoveredPhaseShift); 
	
			// Command aborted
			IF FB_MC2_AxisBasic_M_nMC_PhasingRelative_fbMC2_PhasingRelative.CommandAborted THEN
				FB_MC2_AxisBasic_M_nMC_PhasingRelative_iState:= 030;
			ELSE
				// Error handling
				IF FB_MC2_AxisBasic_M_nMC_PhasingRelative_fbMC2_PhasingRelative.Error THEN
					M_nError(nErrorID:= FB_MC2_AxisBasic_M_nMC_PhasingRelative_fbMC2_PhasingRelative.ErrorID);
					M_nMC_PhasingRelative:= FB_MC2_AxisBasic_M_nMC_PhasingRelative_fbMC2_PhasingRelative.ErrorID;
				ELSE
					// Done
					IF FB_MC2_AxisBasic_M_nMC_PhasingRelative_fbMC2_PhasingRelative.Done THEN
						FB_MC2_AxisBasic_M_nMC_PhasingRelative_iState:= 030;
					END_IF
				END_IF
			END_IF

	030:	// Done
			M_nMC_PhasingRelative:= Tc3_HBI_System.cCOMPLETE;
			
			IF FB_MC2_AxisBasic_M_nMC_PhasingRelative_bExecute THEN
				IF FB_MC2_AxisBasic_M_nMC_PhasingRelative_fbMC2_PhasingRelative.CommandAborted THEN
					M_nMC_PhasingRelative:= Tc3_HBI_System.cABORTED;
				END_IF
			ELSE
				FB_MC2_AxisBasic_M_nMC_PhasingRelative_fbMC2_HaltParsing(Master:= FB_MC2_AxisBasic_M_nMC_PhasingRelative_pMaster^, Slave:= _stAXIS_REF, Execute:= FALSE); 
				FB_MC2_AxisBasic_M_nMC_PhasingRelative_fbMC2_PhasingRelative(Master:= FB_MC2_AxisBasic_M_nMC_PhasingRelative_pMaster^, Slave:= _stAXIS_REF, Execute:= FALSE); 
				FB_MC2_AxisBasic_M_nMC_PhasingRelative_iState:= 000;
			END_IF	

ELSE
	FB_MC2_AxisBasic_M_nMC_PhasingRelative_iState:= 000;
END_CASE
END_METHOD

//	The result of the method is an unsigned double integer
//	0 = idle 
//	1 = coupled
//	2 = starting
//	3 = running
//	4 = aborted
// 	5 = no hardware connected
// 	6 = Spare
//	7 = pointer or index error
//	8 = mapping error
//	9 = parameter error
//	10 = complete
//	Any other number = ErrorID
METHOD PUBLIC M_nMC_PositionLagMonitoring : UDINT
VAR_INPUT
	bEnable: BOOL;
	bDisable: BOOL;
END_VAR
// Local variable
FB_MC2_AxisBasic_M_nMC_PositionLagMonitoring_bEnable:= bEnable;
FB_MC2_AxisBasic_M_nMC_PositionLagMonitoring_bDisable:= bDisable;

// Wait for bEnable or bDisable
IF _stAXIS_REF.NcToPlc.AxisID > 0 THEN
	FB_MC2_AxisBasic_M_nMC_PositionLagMonitoring_fbExecute1_R_TRIG(CLK:= bEnable);
	IF FB_MC2_AxisBasic_M_nMC_PositionLagMonitoring_fbExecute1_R_TRIG.Q THEN
		IF NOT FB_MC2_AxisBasic_M_nMC_PositionLagMonitoring_bDisable THEN
			FB_MC2_AxisBasic_M_nMC_PositionLagMonitoring_nData:= 1;		// TRUE
			FB_MC2_AxisBasic_M_nMC_PositionLagMonitoring_iState:= 001;
		END_IF	
	END_IF
	FB_MC2_AxisBasic_M_nMC_PositionLagMonitoring_fbExecute2_R_TRIG(CLK:= FB_MC2_AxisBasic_M_nMC_PositionLagMonitoring_bDisable);
	IF FB_MC2_AxisBasic_M_nMC_PositionLagMonitoring_fbExecute2_R_TRIG.Q THEN
		IF NOT FB_MC2_AxisBasic_M_nMC_PositionLagMonitoring_bEnable THEN
			FB_MC2_AxisBasic_M_nMC_PositionLagMonitoring_nData:= 0;		// FALSE
			FB_MC2_AxisBasic_M_nMC_PositionLagMonitoring_iState:= 001;
		END_IF	
	END_IF
ELSE
	FB_MC2_AxisBasic_M_nMC_PositionLagMonitoring_fbExecute1_R_TRIG(CLK:= FALSE);
	FB_MC2_AxisBasic_M_nMC_PositionLagMonitoring_fbExecute2_R_TRIG(CLK:= FALSE);
	FB_MC2_AxisBasic_M_nMC_PositionLagMonitoring_iState:= 000;
	IF FB_MC2_AxisBasic_M_nMC_PositionLagMonitoring_bEnable OR FB_MC2_AxisBasic_M_nMC_PositionLagMonitoring_bDisable THEN
		M_nMC_PositionLagMonitoring:= Tc3_HBI_System.cMAPPING_ERROR;
	END_IF
	RETURN;
END_IF


//**********************************
// Main sequence
//**********************************
CASE FB_MC2_AxisBasic_M_nMC_PositionLagMonitoring_iState OF

	000:	// Do nothing

	001:	// Write data
			M_nMC_PositionLagMonitoring:= Tc3_HBI_System.cSTARTING;
			IF _stAXIS_REF.NcToPlc.AxisID > 0 THEN
				FB_MC2_AxisBasic_M_nMC_PositionLagMonitoring_fbADSWrite(LEN:= SIZEOF(FB_MC2_AxisBasic_M_nMC_PositionLagMonitoring_nData), SRCADDR:= ADR(FB_MC2_AxisBasic_M_nMC_PositionLagMonitoring_nData), WRITE:= FALSE); 
				FB_MC2_AxisBasic_M_nMC_PositionLagMonitoring_fbADSWrite(
					NETID:= , 
					PORT:= 501, 
					IDXGRP:= 16#6000 + _stAXIS_REF.NcToPlc.AxisId, 
					IDXOFFS:= 16#10, 
					LEN:= SIZEOF(FB_MC2_AxisBasic_M_nMC_PositionLagMonitoring_nData), 
					SRCADDR:= ADR(FB_MC2_AxisBasic_M_nMC_PositionLagMonitoring_nData), 
					WRITE:= TRUE, 
					TMOUT:= T#2S, 
					BUSY=> , 
					ERR=> , 
					ERRID=> );
			
				FB_MC2_AxisBasic_M_nMC_PositionLagMonitoring_iState:= FB_MC2_AxisBasic_M_nMC_PositionLagMonitoring_iState +1;
			END_IF

	002:	// Write data - Done	
			M_nMC_PositionLagMonitoring:= Tc3_HBI_System.cRUNNING;
			FB_MC2_AxisBasic_M_nMC_PositionLagMonitoring_fbADSWrite(LEN:= SIZEOF(FB_MC2_AxisBasic_M_nMC_PositionLagMonitoring_nData), SRCADDR:= ADR(FB_MC2_AxisBasic_M_nMC_PositionLagMonitoring_nData), WRITE:= TRUE); 
			
			// Error
			IF FB_MC2_AxisBasic_M_nMC_PositionLagMonitoring_fbADSWrite.ERR THEN
				M_nError(nErrorID:= FB_MC2_AxisBasic_M_nMC_PositionLagMonitoring_fbADSWrite.ERRID);
				M_nMC_PositionLagMonitoring:= FB_MC2_AxisBasic_M_nMC_PositionLagMonitoring_fbADSWrite.ERRID;
			ELSE
				// Done
				IF NOT FB_MC2_AxisBasic_M_nMC_PositionLagMonitoring_fbADSWrite.Busy THEN
					FB_MC2_AxisBasic_M_nMC_PositionLagMonitoring_fbADSWrite(LEN:= SIZEOF(FB_MC2_AxisBasic_M_nMC_PositionLagMonitoring_nData), SRCADDR:= ADR(FB_MC2_AxisBasic_M_nMC_PositionLagMonitoring_nData), WRITE:= FALSE); 
					FB_MC2_AxisBasic_M_nMC_PositionLagMonitoring_iState:= FB_MC2_AxisBasic_M_nMC_PositionLagMonitoring_iState +1;
				END_IF
			END_IF

	003:	// Done
			M_nMC_PositionLagMonitoring:= Tc3_HBI_System.cCOMPLETE;

			IF NOT FB_MC2_AxisBasic_M_nMC_PositionLagMonitoring_bEnable AND NOT FB_MC2_AxisBasic_M_nMC_PositionLagMonitoring_bDisable THEN
				FB_MC2_AxisBasic_M_nMC_PositionLagMonitoring_iState:= 000;
			END_IF

ELSE
	FB_MC2_AxisBasic_M_nMC_PositionLagMonitoring_iState:= 000;
END_CASE
END_METHOD

//	The result of the method is an unsigned double integer
//	0 = idle 
//	1 = coupled
//	2 = starting
//	3 = running
//	4 = aborted
// 	5 = no hardware connected
// 	6 = Spare
//	7 = pointer or index error
//	8 = mapping error
//	9 = parameter error
//	10 = complete
//	Any other number = ErrorID
METHOD PUBLIC M_nMC_Power : UDINT
VAR_INPUT
	bEnable: BOOL;
	bE_Stop: BOOL;
	bE_StopDelay: BOOL;
	bEnable_Positive: BOOL;
	bEnable_Negative: BOOL;
END_VAR
// Local variable
FB_MC2_AxisBasic_M_nMC_Power_bEnable:= bEnable;
FB_MC2_AxisBasic_M_nMC_Power_bE_Stop:= bE_Stop;
FB_MC2_AxisBasic_M_nMC_Power_bE_StopDelay:= bE_StopDelay;
FB_MC2_AxisBasic_M_nMC_Power_bEnable_Positive:= bEnable_Positive;
FB_MC2_AxisBasic_M_nMC_Power_bEnable_Negative:= bEnable_Negative; 

//**********************************
// Reset 
//**********************************
IF _bReset THEN
	
	// Reset all methods
	M_nMC_ClrLagError(bExecute:= FB_MC2_AxisBasic_M_nMC_ClrLagError_bExecute);
	M_nMC_DeadTimeComp();
	M_nMC_GearIn(bExecute:= FB_MC2_AxisBasic_M_nMC_GearIn_bExecute, pMaster:= FB_MC2_AxisBasic_M_nMC_GearIn_pMaster, lrRatioNumerator:= FB_MC2_AxisBasic_M_nMC_GearIn_lrRatioNumerator, iRatioDenominator:= FB_MC2_AxisBasic_M_nMC_GearIn_iRatioDenominator);
	M_nMC_GearInDyn(bEnable:= FB_MC2_AxisBasic_M_nMC_GearInDyn_bEnable, pMaster:= FB_MC2_AxisBasic_M_nMC_GearInDyn_pMaster, lrGearRatio:= FB_MC2_AxisBasic_M_nMC_GearInDyn_lrGearRatio);
	M_nMC_GearInMultiMaster(bEnable:= FB_MC2_AxisBasic_M_nMC_GearInMultiMaster_bEnable, pMaster1:= FB_MC2_AxisBasic_M_nMC_GearInMultiMaster_pMaster1, pMaster2:= FB_MC2_AxisBasic_M_nMC_GearInMultiMaster_pMaster2, pMaster3:= FB_MC2_AxisBasic_M_nMC_GearInMultiMaster_pMaster3, pMaster4:= FB_MC2_AxisBasic_M_nMC_GearInMultiMaster_pMaster4);
	M_nMC_GearOut(bExecute:= FB_MC2_AxisBasic_M_nMC_GearOut_bExecute);
	M_nMC_InverseMotor(bExecute:= FB_MC2_AxisBasic_M_nMC_InverseMotor_bExecute, bInverse:= FB_MC2_AxisBasic_M_nMC_InverseMotor_bInverse);
	M_nMC_PhasingAbsolute(bExecute:= FB_MC2_AxisBasic_M_nMC_PhasingAbsolute_bExecute, pMaster:= FB_MC2_AxisBasic_M_nMC_PhasingAbsolute_pMaster, lrPhaseShift:= FB_MC2_AxisBasic_M_nMC_PhasingAbsolute_lrPhaseShift, lrVelocity:= FB_MC2_AxisBasic_M_nMC_PhasingAbsolute_lrVelocity);
	M_nMC_PhasingRelative(bExecute:= FB_MC2_AxisBasic_M_nMC_PhasingRelative_bExecute, pMaster:= FB_MC2_AxisBasic_M_nMC_PhasingRelative_pMaster, lrPhaseShift:= FB_MC2_AxisBasic_M_nMC_PhasingRelative_lrPhaseShift, lrVelocity:= FB_MC2_AxisBasic_M_nMC_PhasingRelative_lrVelocity);
	M_nMC_PositionLagMonitoring(bEnable:= FB_MC2_AxisBasic_M_nMC_PositionLagMonitoring_bEnable, bDisable:= FB_MC2_AxisBasic_M_nMC_PositionLagMonitoring_bDisable);
	M_nMC_ReadParameter();
	M_nMC_RegCorrection(bExecute:= FB_MC2_AxisBasic_M_nMC_RegCorrectiom_bExecute, pRegCorrection:= FB_MC2_AxisBasic_M_nMC_RegCorrectiom_pRegCorrection);	
	M_nMC_SetEncoderOffset(bExecute:= FB_MC2_AxisBasic_M_nMC_SetEncoderOffset_bExecute, lrOffset:= FB_MC2_AxisBasic_M_nMC_SetEncoderOffset_lrOffset);	
	M_nMC_SetFeedConstant(bExecute:= FB_MC2_AxisBasic_M_nMC_SetFeedConstant_bExecute, lrFeedConstant:= FB_MC2_AxisBasic_M_nMC_SetFeedConstant_lrFeedConstant);
	M_nMC_SetModuloFactor(bExecute:= FB_MC2_AxisBasic_M_nMC_SetModuloFactor_bExecute, lrModuloFactor:= FB_MC2_AxisBasic_M_nMC_SetModuloFactor_lrModuloFactor);
	M_nMC_SetPosition(bExecute:= FB_MC2_AxisBasic_M_nMC_SetPosition_bExecute, lrPosition:= FB_MC2_AxisBasic_M_nMC_SetPosition_lrPosition);
	M_nMC_SetPositionRelative(bExecute:= FB_MC2_AxisBasic_M_nMC_SetPositionRelative_bExecute, lrPosition:= FB_MC2_AxisBasic_M_nMC_SetPositionRelative_lrPosition);
	M_nMC_SetScaleFactor(bExecute:= FB_MC2_AxisBasic_M_nMC_SetScaleFactor_bExecute, lrScaleFactor:= FB_MC2_AxisBasic_M_nMC_SetScaleFactor_lrScaleFactor);
	M_nMC_SetVeloKvFactor(bExecute:= FB_MC2_AxisBasic_M_nMC_SetVeloKvFactor_bExecute, lrKvFactor:= FB_MC2_AxisBasic_M_nMC_SetVeloKvFactor_lrKvFactor);
END_IF

// Call methodes
IF _stAXIS_REF.NcToPlc.AxisID > 0 THEN
	FB_MC2_AxisBasic_M_nMC_Power_Status:= SUPER^.M_nMC_Power(bEnable:= FB_MC2_AxisBasic_M_nMC_Power_bEnable, bE_Stop:= FB_MC2_AxisBasic_M_nMC_Power_bE_Stop, bE_StopDelay:= FB_MC2_AxisBasic_M_nMC_Power_bE_StopDelay, bEnable_Positive:= FB_MC2_AxisBasic_M_nMC_Power_bEnable_Positive, bEnable_Negative:= FB_MC2_AxisBasic_M_nMC_Power_bEnable_Negative); 
	M_nMC_ReadParameter();
END_IF


//**********************************
// Error handling
//**********************************
IF _stAXIS_REF.Status.Error THEN
	M_nError(_stAXIS_REF.Status.ErrorID);
	M_nMC_Power:= _nErrorID;
ELSE

	// Method return value
	IF _bError THEN
		M_nMC_Power:= _nErrorID;
	ELSE
		M_nMC_Power:= FB_MC2_AxisBasic_M_nMC_Power_Status;
	END_IF

END_IF
END_METHOD

//	The result of the method is an unsigned double integer
//	0 = idle 
//	1 = coupled
//	2 = starting
//	3 = running
//	4 = aborted
// 	5 = no hardware connected
// 	6 = Spare
//	7 = pointer or index error
//	8 = mapping error
//	9 = parameter error
//	10 = complete
//	Any other number = ErrorID
METHOD PRIVATE M_nMC_ReadParameter : UDINT
VAR_INPUT
END_VAR
//**********************************
// Reset 
//**********************************
IF _bReset THEN
	IF _bError THEN
		IF NOT FB_MC2_AxisBasic_M_nMC_ReadParameter_bDone THEN
			FB_MC2_AxisBasic_M_nMC_ReadParameter_fbADSREAD(READ:= FALSE);
			FB_MC2_AxisBasic_M_nMC_ReadParameter_iState:= 000;
		END_IF
	END_IF
END_IF

//**********************************
// Wait for AxisID
//**********************************
IF _stAXIS_REF.NcToPlc.AxisID > 0 THEN
	FB_MC2_AxisBasic_M_nMC_ReadParameter_fbExecute_R_TRIG(CLK:= TRUE);
	IF FB_MC2_AxisBasic_M_nMC_ReadParameter_fbExecute_R_TRIG.Q THEN
		FB_MC2_AxisBasic_M_nMC_ReadParameter_iState:= 001;
	END_IF
ELSE
	FB_MC2_AxisBasic_M_nMC_ReadParameter_fbExecute_R_TRIG(CLK:= FALSE);
	FB_MC2_AxisBasic_M_nMC_ReadParameter_iState:= 000;
	RETURN;
END_IF


//**********************************
// Main sequence
//**********************************
CASE FB_MC2_AxisBasic_M_nMC_ReadParameter_iState OF

	000: 	// Do nothing

	001:	// Read MaxVelocity
			M_nMC_ReadParameter:= Tc3_HBI_System.cSTARTING;
			FB_MC2_AxisBasic_M_nMC_ReadParameter_fbADSREAD(READ:= FALSE);
			FB_MC2_AxisBasic_M_nMC_ReadParameter_fbADSREAD(
				NETID:= , 
				PORT:= 501, 
				IDXGRP:= 16#4000 + _stAXIS_REF.NcToPlc.AxisId, 
				IDXOFFS:= 16#27, 
				LEN:= SIZEOF(FB_MC2_AxisBasic_M_nMC_ReadParameter_lrTempMaxVelocity), 
				DESTADDR:= ADR(FB_MC2_AxisBasic_M_nMC_ReadParameter_lrTempMaxVelocity), 
				READ:= TRUE, 
				TMOUT:= Tc2_System.DEFAULT_ADS_TIMEOUT, 
				BUSY=> , 
				ERR=> , 
				ERRID=> );
 
			FB_MC2_AxisBasic_M_nMC_ReadParameter_iState:= FB_MC2_AxisBasic_M_nMC_ReadParameter_iState +1;
		
	002:	// Read parameter done	
			M_nMC_ReadParameter:= Tc3_HBI_System.cRUNNING;	
			FB_MC2_AxisBasic_M_nMC_ReadParameter_fbADSREAD(READ:= TRUE);
		
			// Error handling
			IF FB_MC2_AxisBasic_M_nMC_ReadParameter_fbADSREAD.ERR THEN
				M_nError(nErrorID:= FB_MC2_AxisBasic_M_nMC_ReadParameter_fbADSREAD.ERRID);
				M_nMC_ReadParameter:= FB_MC2_AxisBasic_M_nMC_ReadParameter_fbADSREAD.ERRID;
			ELSE
				// Done
				IF NOT FB_MC2_AxisBasic_M_nMC_ReadParameter_fbADSREAD.BUSY THEN
					FB_MC2_AxisBasic_M_nMC_ReadParameter_fbADSREAD(READ:= FALSE); 
					FB_MC2_AxisBasic_M_nMC_ReadParameter_lrMaxVelocity:= FB_MC2_AxisBasic_M_nMC_ReadParameter_lrTempMaxVelocity - 0.0001;			// Offest to max velocity
					FB_MC2_AxisBasic_M_nMC_ReadParameter_iState:= FB_MC2_AxisBasic_M_nMC_ReadParameter_iState +1;
				END_IF
			END_IF
			
	003:	// Done
			M_nMC_ReadParameter:= Tc3_HBI_System.cCOMPLETE;
			FB_MC2_AxisBasic_M_nMC_ReadParameter_bDone:= TRUE;
		
ELSE
	FB_MC2_AxisBasic_M_nMC_ReadParameter_iState:= 000;
END_CASE
END_METHOD

//	The result of the method is an unsigned double integer
//	0 = idle 
//	1 = coupled
//	2 = starting
//	3 = running
//	4 = aborted
// 	5 = no hardware connected
// 	6 = Spare
//	7 = pointer or index error
//	8 = mapping error
//	9 = parameter error
//	10 = complete
//	Any other number = ErrorID
METHOD PUBLIC M_nMC_RegCorrection : UDINT
VAR_INPUT
	bExecute: BOOL;
	pRegCorrection: POINTER TO ST_MC2_RegCorrection;
END_VAR
// Local variable
FB_MC2_AxisBasic_M_nMC_RegCorrectiom_bExecute:= bExecute;
FB_MC2_AxisBasic_M_nMC_RegCorrectiom_pRegCorrection:= pRegCorrection;

//**********************************
// Pointer check
//**********************************
IF FB_MC2_AxisBasic_M_nMC_RegCorrectiom_pRegCorrection = 0 THEN
	IF FB_MC2_AxisBasic_M_nMC_RegCorrectiom_bExecute THEN
		IF _stAXIS_REF.NcToPlc.AxisID > 0 THEN
			FB_MC2_AxisBasic_M_nMC_RegCorrectiom_iState:= 000;
			M_nMC_RegCorrection:= Tc3_HBI_System.cPOINTER_OR_INDEX_ERROR;
		END_IF
	END_IF
	RETURN;
END_IF

//**********************************
// Reset 
//**********************************
IF _bReset THEN
	IF _bError THEN
		FB_MC2_AxisBasic_M_nMC_RegCorrectiom_fbMC2_AbortSuperposition(Execute:= FALSE, Axis:= _stAXIS_REF);
		FB_MC2_AxisBasic_M_nMC_RegCorrectiom_fbMC2_MoveSuperImposed(Axis:= _stAXIS_REF, Execute:= FALSE); 
		FB_MC2_AxisBasic_M_nMC_RegCorrectiom_iState:= 000;
	END_IF
END_IF

//**********************************
// Wait for execute
//**********************************
IF _stAXIS_REF.NcToPlc.AxisID > 0 THEN
	FB_MC2_AxisBasic_M_nMC_RegCorrectiom_fbExecute_R_TRIG(CLK:= FB_MC2_AxisBasic_M_nMC_RegCorrectiom_bExecute);
	IF FB_MC2_AxisBasic_M_nMC_RegCorrectiom_fbExecute_R_TRIG.Q THEN
		FB_MC2_AxisBasic_M_nMC_RegCorrectiom_fbMC2_AbortSuperposition(Execute:= FALSE, Axis:= _stAXIS_REF);
		FB_MC2_AxisBasic_M_nMC_RegCorrectiom_fbMC2_MoveSuperImposed(Axis:= _stAXIS_REF, Execute:= FALSE); 
		FB_MC2_AxisBasic_M_nMC_RegCorrectiom_iState:= 010;
	END_IF
	FB_MC2_AxisBasic_M_nMC_RegCorrectiom_fbNotExecute_R_TRIG(CLK:= NOT FB_MC2_AxisBasic_M_nMC_RegCorrectiom_bExecute);
	IF FB_MC2_AxisBasic_M_nMC_RegCorrectiom_fbNotExecute_R_TRIG.Q THEN
		IF _stAXIS_REF.NcToPlc.AxisID > 0 THEN
			FB_MC2_AxisBasic_M_nMC_RegCorrectiom_fbMC2_AbortSuperposition(Execute:= FALSE, Axis:= _stAXIS_REF);
			FB_MC2_AxisBasic_M_nMC_RegCorrectiom_fbMC2_MoveSuperImposed(Axis:= _stAXIS_REF, Execute:= FALSE); 
			IF FB_MC2_AxisBasic_M_nMC_RegCorrectiom_fbMC2_MoveSuperImposed.Busy THEN
				FB_MC2_AxisBasic_M_nMC_RegCorrectiom_iState:= 001;
			ELSE
				FB_MC2_AxisBasic_M_nMC_RegCorrectiom_iState:= 000;
			END_IF
		END_IF	
	END_IF
ELSE
	FB_MC2_AxisBasic_M_nMC_RegCorrectiom_fbExecute_R_TRIG(CLK:= FALSE);
	FB_MC2_AxisBasic_M_nMC_RegCorrectiom_fbNotExecute_R_TRIG(CLK:= FALSE);
	FB_MC2_AxisBasic_M_nMC_RegCorrectiom_iState:= 000;
	IF FB_MC2_AxisBasic_M_nMC_RegCorrectiom_bExecute THEN
		M_nMC_RegCorrection:= Tc3_HBI_System.cMAPPING_ERROR;
	END_IF
	RETURN;
END_IF


//**********************************
// Main sequence
//**********************************
CASE FB_MC2_AxisBasic_M_nMC_RegCorrectiom_iState OF

	000: 	// Do nothing
	
	001:	// Abort Superposition
			M_nMC_RegCorrection:= Tc3_HBI_System.cSTARTING;
			FB_MC2_AxisBasic_M_nMC_RegCorrectiom_fbMC2_AbortSuperposition(Execute:= FALSE, Axis:= _stAXIS_REF);
			FB_MC2_AxisBasic_M_nMC_RegCorrectiom_fbMC2_AbortSuperposition(
				Execute:= TRUE, 
				Done=> , 
				Busy=> , 
				Error=> , 
				ErrorID=> , 
				Axis:= _stAXIS_REF);
	
			FB_MC2_AxisBasic_M_nMC_RegCorrectiom_iState:= FB_MC2_AxisBasic_M_nMC_RegCorrectiom_iState +1;	
				
	002:	// Abort Superposition - Done
			M_nMC_RegCorrection:= Tc3_HBI_System.cRUNNING;
			FB_MC2_AxisBasic_M_nMC_RegCorrectiom_fbMC2_AbortSuperposition(Execute:= TRUE, Axis:= _stAXIS_REF);

			// Error handling
			IF FB_MC2_AxisBasic_M_nMC_RegCorrectiom_fbMC2_AbortSuperposition.Error THEN
				IF FB_MC2_AxisBasic_M_nMC_RegCorrectiom_fbMC2_AbortSuperposition.ErrorID <> 16966 THEN
					M_nError(nErrorID:= FB_MC2_AxisBasic_M_nMC_RegCorrectiom_fbMC2_AbortSuperposition.ErrorID);
					M_nMC_RegCorrection:= FB_MC2_AxisBasic_M_nMC_RegCorrectiom_fbMC2_AbortSuperposition.ErrorID;
				ELSE
					FB_MC2_AxisBasic_M_nMC_RegCorrectiom_fbMC2_AbortSuperposition(Execute:= FALSE, Axis:= _stAXIS_REF);
					FB_MC2_AxisBasic_M_nMC_RegCorrectiom_iState:= 000;	
				END_IF	
			ELSE
				// Done
				IF FB_MC2_AxisBasic_M_nMC_RegCorrectiom_fbMC2_AbortSuperposition.Done THEN
					FB_MC2_AxisBasic_M_nMC_RegCorrectiom_fbMC2_AbortSuperposition(Execute:= FALSE, Axis:= _stAXIS_REF);
					FB_MC2_AxisBasic_M_nMC_RegCorrectiom_iState:= 000;	
				END_IF
			END_IF
		
	010:	// MoveSuperImposed
			M_nMC_RegCorrection:= Tc3_HBI_System.cRUNNING;
			FB_MC2_AxisBasic_M_nMC_RegCorrectiom_fbMC2_MoveSuperImposed(Axis:= _stAXIS_REF, Execute:= FALSE); 
			FB_MC2_AxisBasic_M_nMC_RegCorrectiom_fbMC2_MoveSuperImposed(
				Axis:= _stAXIS_REF, 
				Execute:= TRUE, 
				Mode:= FB_MC2_AxisBasic_M_nMC_RegCorrectiom_pRegCorrection^.Set.eMode, 
				Distance:= FB_MC2_AxisBasic_M_nMC_RegCorrectiom_pRegCorrection^.Set.lrDistance, 
				VelocityDiff:= FB_MC2_AxisBasic_M_nMC_RegCorrectiom_pRegCorrection^.Set.lrVelocityDiff, 
				Acceleration:= FB_MC2_AxisBasic_M_nMC_RegCorrectiom_pRegCorrection^.Set.lrAcceleration, 
				Deceleration:= FB_MC2_AxisBasic_M_nMC_RegCorrectiom_pRegCorrection^.Set.lrDeceleration, 
				Jerk:= FB_MC2_AxisBasic_M_nMC_RegCorrectiom_pRegCorrection^.Set.lrJerk, 
				VelocityProcess:= FB_MC2_AxisBasic_M_nMC_RegCorrectiom_pRegCorrection^.Set.lrVelocityProcess, 
				Length:= FB_MC2_AxisBasic_M_nMC_RegCorrectiom_pRegCorrection^.Set.lrLength, 
				Options:= FB_MC2_AxisBasic_M_nMC_RegCorrectiom_pRegCorrection^.Set.eOptions, 
				Done=> , 
				Busy=> , 
				Active=> , 
				CommandAborted=> , 
				Error=> , 
				ErrorID=> , 
				Warning=> FB_MC2_AxisBasic_M_nMC_RegCorrectiom_pRegCorrection^.Get.bWarning, 
				WarningId=> FB_MC2_AxisBasic_M_nMC_RegCorrectiom_pRegCorrection^.Get.nWarningId, 
				ActualVelocityDiff=> FB_MC2_AxisBasic_M_nMC_RegCorrectiom_pRegCorrection^.Get.lrActualVelocityDiff, 
				ActualDistance=> FB_MC2_AxisBasic_M_nMC_RegCorrectiom_pRegCorrection^.Get.lrActualDistance, 
				ActualLength=> FB_MC2_AxisBasic_M_nMC_RegCorrectiom_pRegCorrection^.Get.lrActualLength, 
				ActualAcceleration=> FB_MC2_AxisBasic_M_nMC_RegCorrectiom_pRegCorrection^.Get.lrActualAcceleration, 
				ActualDeceleration=> FB_MC2_AxisBasic_M_nMC_RegCorrectiom_pRegCorrection^.Get.lrActualDeceleration);
	
			FB_MC2_AxisBasic_M_nMC_RegCorrectiom_iState:= FB_MC2_AxisBasic_M_nMC_RegCorrectiom_iState +1;
			
	011:	// Done 
			M_nMC_RegCorrection:= Tc3_HBI_System.cRUNNING;
			FB_MC2_AxisBasic_M_nMC_RegCorrectiom_fbMC2_MoveSuperImposed(
				Axis:= _stAXIS_REF, 
				Execute:= TRUE, 
				Done=> , 
				Busy=> , 
				Active=> , 
				CommandAborted=> , 
				Error=> , 
				ErrorID=> , 
				Warning=> FB_MC2_AxisBasic_M_nMC_RegCorrectiom_pRegCorrection^.Get.bWarning, 
				WarningId=> FB_MC2_AxisBasic_M_nMC_RegCorrectiom_pRegCorrection^.Get.nWarningId, 
				ActualVelocityDiff=> FB_MC2_AxisBasic_M_nMC_RegCorrectiom_pRegCorrection^.Get.lrActualVelocityDiff, 
				ActualDistance=> FB_MC2_AxisBasic_M_nMC_RegCorrectiom_pRegCorrection^.Get.lrActualDistance, 
				ActualLength=> FB_MC2_AxisBasic_M_nMC_RegCorrectiom_pRegCorrection^.Get.lrActualLength, 
				ActualAcceleration=> FB_MC2_AxisBasic_M_nMC_RegCorrectiom_pRegCorrection^.Get.lrActualAcceleration, 
				ActualDeceleration=> FB_MC2_AxisBasic_M_nMC_RegCorrectiom_pRegCorrection^.Get.lrActualDeceleration);

			// Command aborted
			IF FB_MC2_AxisBasic_M_nMC_RegCorrectiom_fbMC2_MoveSuperImposed.CommandAborted THEN
				FB_MC2_AxisBasic_M_nMC_RegCorrectiom_iState:= 030;
			ELSE
				// Error handling
				IF FB_MC2_AxisBasic_M_nMC_RegCorrectiom_fbMC2_MoveSuperImposed.Error THEN
					M_nError(nErrorID:= FB_MC2_AxisBasic_M_nMC_RegCorrectiom_fbMC2_MoveSuperImposed.ErrorID);
					M_nMC_RegCorrection:= FB_MC2_AxisBasic_M_nMC_RegCorrectiom_fbMC2_MoveSuperImposed.ErrorID;
				ELSE
					// Done
					IF FB_MC2_AxisBasic_M_nMC_RegCorrectiom_fbMC2_MoveSuperImposed.Done THEN
						FB_MC2_AxisBasic_M_nMC_RegCorrectiom_iState:= 030;
					END_IF
				END_IF
			END_IF

	030:	// Done
			M_nMC_RegCorrection:= Tc3_HBI_System.cCOMPLETE;
			
			IF FB_MC2_AxisBasic_M_nMC_RegCorrectiom_bExecute THEN
				IF FB_MC2_AxisBasic_M_nMC_RegCorrectiom_fbMC2_MoveSuperImposed.CommandAborted THEN
					M_nMC_RegCorrection:= Tc3_HBI_System.cABORTED;
				END_IF
			ELSE
				FB_MC2_AxisBasic_M_nMC_RegCorrectiom_fbMC2_AbortSuperposition(Execute:= FALSE, Axis:= _stAXIS_REF);
				FB_MC2_AxisBasic_M_nMC_RegCorrectiom_fbMC2_MoveSuperImposed(Axis:= _stAXIS_REF, Execute:= FALSE); 
				FB_MC2_AxisBasic_M_nMC_RegCorrectiom_iState:= 000;
			END_IF	

ELSE
	FB_MC2_AxisBasic_M_nMC_RegCorrectiom_iState:= 000;
END_CASE
END_METHOD

//	The result of the method is an unsigned double integer
//	0 = idle 
//	1 = coupled
//	2 = starting
//	3 = running
//	4 = aborted
// 	5 = no hardware connected
// 	6 = Spare
//	7 = pointer or index error
//	8 = mapping error
//	9 = parameter error
//	10 = complete
//	Any other number = ErrorID
METHOD PUBLIC M_nMC_SetEncoderOffset : UDINT
VAR_INPUT
	bExecute: BOOL;
	lrOffset: LREAL;
END_VAR
// Local variable
FB_MC2_AxisBasic_M_nMC_SetEncoderOffset_bExecute:= bExecute;
FB_MC2_AxisBasic_M_nMC_SetEncoderOffset_lrOffset:= lrOffset;

//**********************************
// Reset 
//**********************************
IF _bReset THEN
	IF _bError THEN
		FB_MC2_AxisBasic_M_nMC_SetEncoderOffset_fbADSWRITE(WRITE:= FALSE); 
		FB_MC2_AxisBasic_M_nMC_SetEncoderOffset_fbExecute_R_TRIG(CLK:= FALSE);
		FB_MC2_AxisBasic_M_nMC_SetEncoderOffset_iState:= 000;
	END_IF
END_IF

//**********************************
// Wait for execute
//**********************************
IF _stAXIS_REF.NcToPlc.AxisID > 0 THEN
	FB_MC2_AxisBasic_M_nMC_SetEncoderOffset_fbExecute_R_TRIG(CLK:= FB_MC2_AxisBasic_M_nMC_SetEncoderOffset_bExecute);
	IF FB_MC2_AxisBasic_M_nMC_SetEncoderOffset_fbExecute_R_TRIG.Q THEN
		FB_MC2_AxisBasic_M_nMC_SetEncoderOffset_iState:= 001;
	END_IF
ELSE
	FB_MC2_AxisBasic_M_nMC_SetEncoderOffset_fbExecute_R_TRIG(CLK:= FALSE);
	FB_MC2_AxisBasic_M_nMC_SetEncoderOffset_iState:= 000;
	M_nMC_SetEncoderOffset:= Tc3_HBI_System.cPARAMETER_ERROR;
	IF FB_MC2_AxisBasic_M_nMC_SetEncoderOffset_bExecute THEN
		M_nMC_SetEncoderOffset:= Tc3_HBI_System.cMAPPING_ERROR;
	END_IF
	RETURN;
END_IF


//**********************************
// Main sequence
//**********************************
CASE FB_MC2_AxisBasic_M_nMC_SetEncoderOffset_iState OF

	000: 	// Do nothing

	001:	// Set Encoder offset
			M_nMC_SetEncoderOffset:= Tc3_HBI_System.cSTARTING;
			FB_MC2_AxisBasic_M_nMC_SetEncoderOffset_fbADSWRITE(WRITE:= FALSE);
			FB_MC2_AxisBasic_M_nMC_SetEncoderOffset_fbADSWRITE(
				NETID:= '', 
				PORT:= 501, 
				IDXGRP:= 16#5000 + _stAXIS_REF.NcToPlc.AxisId, 
				IDXOFFS:= 16#07, 
				LEN:= SIZEOF(FB_MC2_AxisBasic_M_nMC_SetEncoderOffset_lrOffset), 
				SRCADDR:= ADR(FB_MC2_AxisBasic_M_nMC_SetEncoderOffset_lrOffset), 
				WRITE:= TRUE, 
				TMOUT:= Tc2_System.DEFAULT_ADS_TIMEOUT, 
				BUSY=> , 
				ERR=> , 
				ERRID=> );
 
			FB_MC2_AxisBasic_M_nMC_SetEncoderOffset_iState:= FB_MC2_AxisBasic_M_nMC_SetEncoderOffset_iState +1;
		
	002:	// Done	
			M_nMC_SetEncoderOffset:= Tc3_HBI_System.cRUNNING;	
			FB_MC2_AxisBasic_M_nMC_SetEncoderOffset_fbADSWRITE(WRITE:= TRUE);
		
			// Error handling
			IF FB_MC2_AxisBasic_M_nMC_SetEncoderOffset_fbADSWRITE.ERR THEN
				M_nError(nErrorID:= FB_MC2_AxisBasic_M_nMC_SetEncoderOffset_fbADSWRITE.ERRID);
				M_nMC_SetEncoderOffset:= FB_MC2_AxisBasic_M_nMC_SetEncoderOffset_fbADSWRITE.ERRID;
			ELSE
				// Done
				IF NOT FB_MC2_AxisBasic_M_nMC_SetEncoderOffset_fbADSWRITE.BUSY THEN
					FB_MC2_AxisBasic_M_nMC_SetEncoderOffset_fbADSWRITE(WRITE:= FALSE); 
					FB_MC2_AxisBasic_M_nMC_SetEncoderOffset_iState:= FB_MC2_AxisBasic_M_nMC_SetEncoderOffset_iState +1;
				END_IF
			END_IF
			
	003:	// Done
			M_nMC_SetEncoderOffset:= Tc3_HBI_System.cCOMPLETE;
			IF NOT FB_MC2_AxisBasic_M_nMC_SetEncoderOffset_bExecute THEN	
				FB_MC2_AxisBasic_M_nMC_SetEncoderOffset_iState:= 000;
			END_IF	
		
ELSE
	FB_MC2_AxisBasic_M_nMC_SetEncoderOffset_iState:= 000;
END_CASE
END_METHOD

//	The result of the method is an unsigned double integer
//	0 = idle 
//	1 = coupled
//	2 = starting
//	3 = running
//	4 = aborted
// 	5 = no hardware connected
// 	6 = Spare
//	7 = pointer or index error
//	8 = mapping error
//	9 = parameter error
//	10 = complete
//	Any other number = ErrorID
METHOD PUBLIC M_nMC_SetFeedConstant : UDINT
VAR_INPUT
	bExecute: BOOL;
	lrFeedConstant: LREAL;
END_VAR
// Local variable
FB_MC2_AxisBasic_M_nMC_SetFeedConstant_bExecute:= bExecute;
FB_MC2_AxisBasic_M_nMC_SetFeedConstant_lrFeedConstant:= lrFeedConstant;

//**********************************
// Reset 
//**********************************
IF _bReset THEN
	IF _bError THEN
		FB_MC2_AxisBasic_M_nMC_SetFeedConstant_fbADSWRITE(WRITE:= FALSE); 
		FB_MC2_AxisBasic_M_nMC_SetFeedConstant_fbExecute_R_TRIG(CLK:= FALSE);
		FB_MC2_AxisBasic_M_nMC_SetFeedConstant_iState:= 000;
	END_IF
END_IF

//**********************************
// Parameter check 
//**********************************
IF FB_MC2_AxisBasic_M_nMC_SetFeedConstant_bExecute THEN
	IF FB_MC2_AxisBasic_M_nMC_SetFeedConstant_lrFeedConstant <= 0.0 THEN
		FB_MC2_AxisBasic_M_nMC_SetFeedConstant_fbADSWRITE(WRITE:= FALSE); 
		FB_MC2_AxisBasic_M_nMC_SetFeedConstant_fbExecute_R_TRIG(CLK:= FALSE);
		FB_MC2_AxisBasic_M_nMC_SetFeedConstant_iState:= 000;
		M_nMC_SetFeedConstant:= Tc3_HBI_System.cPARAMETER_ERROR;
		RETURN;
	END_IF
END_IF

//**********************************
// Wait for execute
//**********************************
IF _stAXIS_REF.NcToPlc.AxisID > 0 THEN
	FB_MC2_AxisBasic_M_nMC_SetFeedConstant_fbExecute_R_TRIG(CLK:= FB_MC2_AxisBasic_M_nMC_SetFeedConstant_bExecute);
	IF FB_MC2_AxisBasic_M_nMC_SetFeedConstant_fbExecute_R_TRIG.Q THEN
		FB_MC2_AxisBasic_M_nMC_SetFeedConstant_iState:= 001;
	END_IF
ELSE
	FB_MC2_AxisBasic_M_nMC_SetFeedConstant_fbExecute_R_TRIG(CLK:= FALSE);
	FB_MC2_AxisBasic_M_nMC_SetFeedConstant_iState:= 000;
	IF FB_MC2_AxisBasic_M_nMC_SetFeedConstant_bExecute THEN
		M_nMC_SetFeedConstant:= Tc3_HBI_System.cMAPPING_ERROR;
	END_IF
	RETURN;
END_IF


//**********************************
// Main sequence
//**********************************
CASE FB_MC2_AxisBasic_M_nMC_SetFeedConstant_iState OF

	000: 	// Do nothing

	001:	// Set Feed constant
			M_nMC_SetFeedConstant:= Tc3_HBI_System.cSTARTING;
			FB_MC2_AxisBasic_M_nMC_SetFeedConstant_fbADSWRITE(WRITE:= FALSE);
			FB_MC2_AxisBasic_M_nMC_SetFeedConstant_fbADSWRITE(
				NETID:= '', 
				PORT:= 501, 
				IDXGRP:= 16#5000 + _stAXIS_REF.NcToPlc.AxisId, 
				IDXOFFS:= 16#23, 
				LEN:= SIZEOF(FB_MC2_AxisBasic_M_nMC_SetFeedConstant_lrFeedConstant), 
				SRCADDR:= ADR(FB_MC2_AxisBasic_M_nMC_SetFeedConstant_lrFeedConstant), 
				WRITE:= TRUE, 
				TMOUT:= Tc2_System.DEFAULT_ADS_TIMEOUT, 
				BUSY=> , 
				ERR=> , 
				ERRID=> );
 
			FB_MC2_AxisBasic_M_nMC_SetFeedConstant_iState:= FB_MC2_AxisBasic_M_nMC_SetFeedConstant_iState +1;
		
	002:	// Done	
			M_nMC_SetFeedConstant:= Tc3_HBI_System.cRUNNING;	
			FB_MC2_AxisBasic_M_nMC_SetFeedConstant_fbADSWRITE(WRITE:= TRUE);
		
			// Error handling
			IF FB_MC2_AxisBasic_M_nMC_SetFeedConstant_fbADSWRITE.ERR THEN
				M_nError(nErrorID:= FB_MC2_AxisBasic_M_nMC_SetFeedConstant_fbADSWRITE.ERRID);
				M_nMC_SetFeedConstant:= FB_MC2_AxisBasic_M_nMC_SetFeedConstant_fbADSWRITE.ERRID;
			ELSE
				// Done
				IF NOT FB_MC2_AxisBasic_M_nMC_SetFeedConstant_fbADSWRITE.BUSY THEN
					FB_MC2_AxisBasic_M_nMC_SetFeedConstant_fbADSWRITE(WRITE:= FALSE); 
					FB_MC2_AxisBasic_M_nMC_SetFeedConstant_iState:= FB_MC2_AxisBasic_M_nMC_SetFeedConstant_iState +1;
				END_IF
			END_IF
			
	003:	// Done
			M_nMC_SetFeedConstant:= Tc3_HBI_System.cCOMPLETE;
			IF NOT FB_MC2_AxisBasic_M_nMC_SetFeedConstant_bExecute THEN	
				FB_MC2_AxisBasic_M_nMC_SetFeedConstant_iState:= 000;
			END_IF	
		
ELSE
	FB_MC2_AxisBasic_M_nMC_SetFeedConstant_iState:= 000;
END_CASE
END_METHOD

//	The result of the method is an unsigned double integer
//	0 = idle 
//	1 = coupled
//	2 = starting
//	3 = running
//	4 = aborted
// 	5 = no hardware connected
// 	6 = Spare
//	7 = pointer or index error
//	8 = mapping error
//	9 = parameter error
//	10 = complete
//	Any other number = ErrorID
METHOD PUBLIC M_nMC_SetModuloFactor : UDINT
VAR_INPUT
	bExecute: BOOL;
	lrModuloFactor: LREAL;
END_VAR
// Local variable
FB_MC2_AxisBasic_M_nMC_SetModuloFactor_bExecute:= bExecute;
FB_MC2_AxisBasic_M_nMC_SetModuloFactor_lrModuloFactor:= lrModuloFactor;

//**********************************
// Reset 
//**********************************
IF _bReset THEN
	IF _bError THEN
		FB_MC2_AxisBasic_M_nMC_SetModuloFactor_fbADSWRITE(WRITE:= FALSE); 
		FB_MC2_AxisBasic_M_nMC_SetModuloFactor_iState:= 000;
	END_IF
END_IF

//**********************************
// Parameter check 
//**********************************
IF FB_MC2_AxisBasic_M_nMC_SetModuloFactor_bExecute THEN
	IF FB_MC2_AxisBasic_M_nMC_SetModuloFactor_lrModuloFactor <= 0.0 THEN
		M_nMC_SetModuloFactor:= Tc3_HBI_System.cPARAMETER_ERROR;
		RETURN;
	END_IF	
END_IF


//**********************************
// Wait for execute
//**********************************
IF _stAXIS_REF.NcToPlc.AxisID > 0 THEN
	FB_MC2_AxisBasic_M_nMC_SetModuloFactor_fbExecute_R_TRIG(CLK:= FB_MC2_AxisBasic_M_nMC_SetModuloFactor_bExecute);
	IF FB_MC2_AxisBasic_M_nMC_SetModuloFactor_fbExecute_R_TRIG.Q THEN
		FB_MC2_AxisBasic_M_nMC_SetModuloFactor_iState:= 001;
	END_IF
ELSE
	FB_MC2_AxisBasic_M_nMC_SetModuloFactor_fbExecute_R_TRIG(CLK:= FALSE);
	FB_MC2_AxisBasic_M_nMC_SetModuloFactor_iState:= 000;
	IF FB_MC2_AxisBasic_M_nMC_SetModuloFactor_bExecute THEN
		M_nMC_SetModuloFactor:= Tc3_HBI_System.cMAPPING_ERROR;
	END_IF
	RETURN;
END_IF


//**********************************
// Main sequence
//**********************************
CASE FB_MC2_AxisBasic_M_nMC_SetModuloFactor_iState OF

	000: 	// Do nothing

	001:	// Set Encoder offset
			IF FB_MC2_AxisBasic_M_nMC_SetModuloFactor_bExecute THEN				
				IF FB_MC2_AxisBasic_M_nMC_SetModuloFactor_lrModuloFactor = 0.0 THEN
					M_nMC_SetModuloFactor:= Tc3_HBI_System.cPARAMETER_ERROR;
				ELSE
					M_nMC_SetModuloFactor:= Tc3_HBI_System.cSTARTING;
					FB_MC2_AxisBasic_M_nMC_SetModuloFactor_fbADSWRITE(WRITE:= FALSE);
					FB_MC2_AxisBasic_M_nMC_SetModuloFactor_fbADSWRITE(
						NETID:= '', 
						PORT:= 501, 
						IDXGRP:= 16#5000 + _stAXIS_REF.NcToPlc.AxisId, 
						IDXOFFS:= 16#09, 
						LEN:= SIZEOF(FB_MC2_AxisBasic_M_nMC_SetModuloFactor_lrModuloFactor), 
						SRCADDR:= ADR(FB_MC2_AxisBasic_M_nMC_SetModuloFactor_lrModuloFactor), 
						WRITE:= TRUE, 
						TMOUT:= Tc2_System.DEFAULT_ADS_TIMEOUT, 
						BUSY=> , 
						ERR=> , 
						ERRID=> );
		 
					FB_MC2_AxisBasic_M_nMC_SetModuloFactor_iState:= FB_MC2_AxisBasic_M_nMC_SetModuloFactor_iState +1;
				END_IF
			ELSE
				FB_MC2_AxisBasic_M_nMC_SetModuloFactor_iState:= 000;
			END_IF	
	
	002:	// Done	
			M_nMC_SetModuloFactor:= Tc3_HBI_System.cRUNNING;	
			FB_MC2_AxisBasic_M_nMC_SetModuloFactor_fbADSWRITE(WRITE:= TRUE);
		
			// Error handling
			IF FB_MC2_AxisBasic_M_nMC_SetModuloFactor_fbADSWRITE.ERR THEN
				M_nError(nErrorID:= FB_MC2_AxisBasic_M_nMC_SetModuloFactor_fbADSWRITE.ERRID);
				M_nMC_SetModuloFactor:= FB_MC2_AxisBasic_M_nMC_SetModuloFactor_fbADSWRITE.ERRID;
			ELSE
				// Done
				IF NOT FB_MC2_AxisBasic_M_nMC_SetModuloFactor_fbADSWRITE.BUSY THEN
					FB_MC2_AxisBasic_M_nMC_SetModuloFactor_fbADSWRITE(WRITE:= FALSE); 
					FB_MC2_AxisBasic_M_nMC_SetModuloFactor_iState:= FB_MC2_AxisBasic_M_nMC_SetModuloFactor_iState +1;
				END_IF
			END_IF
			
	003:	// Done
			M_nMC_SetModuloFactor:= Tc3_HBI_System.cCOMPLETE;
			
			IF NOT FB_MC2_AxisBasic_M_nMC_SetModuloFactor_bExecute THEN	
				FB_MC2_AxisBasic_M_nMC_SetModuloFactor_iState:= 000;
			END_IF	
		
ELSE
	FB_MC2_AxisBasic_M_nMC_SetModuloFactor_iState:= 000;
END_CASE
END_METHOD

//	The result of the method is an unsigned double integer
//	0 = idle 
//	1 = coupled
//	2 = starting
//	3 = running
//	4 = aborted
// 	5 = no hardware connected
// 	6 = Spare
//	7 = pointer or index error
//	8 = mapping error
//	9 = parameter error
//	10 = complete
//	Any other number = ErrorID
METHOD PUBLIC M_nMC_SetPosition : UDINT
VAR_INPUT
	bExecute: BOOL;
	lrPosition: LREAL;
END_VAR
// Local variable
FB_MC2_AxisBasic_M_nMC_SetPosition_bExecute:= bExecute;
FB_MC2_AxisBasic_M_nMC_SetPosition_lrPosition:= lrPosition;

//**********************************
// Reset 
//**********************************
IF _bReset THEN
	IF _bError THEN
		FB_MC2_AxisBasic_M_nMC_SetPosition_fbMC2_SetPosition(Axis:= _stAXIS_REF, Execute:= FALSE); 
		FB_MC2_AxisBasic_M_nMC_SetPosition_iState:= 000;
	END_IF
END_IF

//**********************************
// Wait for execute
//**********************************
IF _stAXIS_REF.NcToPlc.AxisID > 0 THEN
	FB_MC2_AxisBasic_M_nMC_SetPosition_fbExecute_R_TRIG(CLK:= FB_MC2_AxisBasic_M_nMC_SetPosition_bExecute);
	IF FB_MC2_AxisBasic_M_nMC_SetPosition_fbExecute_R_TRIG.Q THEN
		FB_MC2_AxisBasic_M_nMC_SetPosition_fbMC2_SetPosition(Axis:= _stAXIS_REF, Execute:= FALSE, Position:= FB_MC2_AxisBasic_M_nMC_SetPosition_lrPosition,  Mode:= FALSE); 
		
		// Axis not coupled	
		IF NOT _stAXIS_REF.Status.Coupled THEN
			FB_MC2_AxisBasic_M_nMC_SetPosition_iState:= 001;
		ELSE
			FB_MC2_AxisBasic_M_nMC_SetPosition_iState:= 010;
		END_IF
	END_IF
ELSE
	FB_MC2_AxisBasic_M_nMC_SetPosition_fbExecute_R_TRIG(CLK:= FALSE);
	FB_MC2_AxisBasic_M_nMC_SetPosition_iState:= 000;
	IF FB_MC2_AxisBasic_M_nMC_SetPosition_bExecute THEN
		M_nMC_SetPosition:= Tc3_HBI_System.cMAPPING_ERROR;
	END_IF
	RETURN;
END_IF


//**********************************
// Main sequence
//**********************************
CASE FB_MC2_AxisBasic_M_nMC_SetPosition_iState OF

	000: 	// Do nothing
	
	001:	// Set Axis position
			M_nMC_SetPosition:= Tc3_HBI_System.cRUNNING;
			IF _stAXIS_REF.NcToPlc.AxisID > 0 THEN
				FB_MC2_AxisBasic_M_nMC_SetPosition_fbMC2_SetPosition(Axis:= _stAXIS_REF, Execute:= FALSE); 
				FB_MC2_AxisBasic_M_nMC_SetPosition_fbMC2_SetPosition(Axis:= _stAXIS_REF, Execute:= TRUE, Position:= FB_MC2_AxisBasic_M_nMC_SetPosition_lrPosition); 
				FB_MC2_AxisBasic_M_nMC_SetPosition_iState:= FB_MC2_AxisBasic_M_nMC_SetPosition_iState +1;
			END_IF
			
	002:	// Set Axis position - Done
			M_nMC_SetPosition:= Tc3_HBI_System.cRUNNING;
			FB_MC2_AxisBasic_M_nMC_SetPosition_fbMC2_SetPosition(Axis:= _stAXIS_REF, Execute:= TRUE); 
			
			// Error handling
			IF FB_MC2_AxisBasic_M_nMC_SetPosition_fbMC2_SetPosition.Error THEN
				M_nError(FB_MC2_AxisBasic_M_nMC_SetPosition_fbMC2_SetPosition.ErrorID);
				M_nMC_SetPosition:= FB_MC2_AxisBasic_M_nMC_SetPosition_fbMC2_SetPosition.ErrorID;
			ELSE
				// Done
				IF FB_MC2_AxisBasic_M_nMC_SetPosition_fbMC2_SetPosition.Done THEN
					FB_MC2_AxisBasic_M_nMC_SetPosition_fbMC2_SetPosition(Axis:= _stAXIS_REF, Execute:= FALSE); 
					FB_MC2_AxisBasic_M_nMC_SetPosition_iState:= 020;
				END_IF
			END_IF
		
	010:	// Coupled
			M_nMC_SetPosition:= Tc3_HBI_System.cCOUPLED;
			IF NOT FB_MC2_AxisBasic_M_nMC_SetPosition_bExecute THEN
				FB_MC2_AxisBasic_M_nMC_SetPosition_fbMC2_SetPosition(Axis:= _stAXIS_REF, Execute:= FALSE); 
				FB_MC2_AxisBasic_M_nMC_SetPosition_iState:= 000;
			END_IF	

	020:	// Done
			M_nMC_SetPosition:= Tc3_HBI_System.cCOMPLETE;
			
			IF NOT FB_MC2_AxisBasic_M_nMC_SetPosition_bExecute THEN
				FB_MC2_AxisBasic_M_nMC_SetPosition_fbMC2_SetPosition(Axis:= _stAXIS_REF, Execute:= FALSE); 
				FB_MC2_AxisBasic_M_nMC_SetPosition_iState:= 000;
			END_IF	
		
ELSE
	FB_MC2_AxisBasic_M_nMC_SetPosition_iState:= 000;
END_CASE
END_METHOD

//	The result of the method is an unsigned double integer
//	0 = idle 
//	1 = coupled
//	2 = starting
//	3 = running
//	4 = aborted
// 	5 = no hardware connected
// 	6 = Spare
//	7 = pointer or index error
//	8 = mapping error
//	9 = parameter error
//	10 = complete
//	Any other number = ErrorID
METHOD PUBLIC M_nMC_SetPositionRelative : UDINT
VAR_INPUT
	bExecute: BOOL;
	lrPosition: LREAL;
END_VAR
// Local variable
FB_MC2_AxisBasic_M_nMC_SetPositionRelative_bExecute:= bExecute;
FB_MC2_AxisBasic_M_nMC_SetPositionRelative_lrPosition:= lrPosition;

//**********************************
// Reset 
//**********************************
IF _bReset THEN
	IF _bError THEN
		FB_MC2_AxisBasic_M_nMC_SetPositionRelative_fbMC2_SetPosition(Axis:= _stAXIS_REF, Execute:= FALSE); 
		FB_MC2_AxisBasic_M_nMC_SetPositionRelative_iState:= 000;
	END_IF
END_IF

//**********************************
// Wait for execute
//**********************************
IF _stAXIS_REF.NcToPlc.AxisID > 0 THEN
	FB_MC2_AxisBasic_M_nMC_SetPositionRelative_fbExecute_R_TRIG(CLK:= FB_MC2_AxisBasic_M_nMC_SetPositionRelative_bExecute);
	IF FB_MC2_AxisBasic_M_nMC_SetPositionRelative_fbExecute_R_TRIG.Q THEN
		FB_MC2_AxisBasic_M_nMC_SetPositionRelative_fbMC2_SetPosition(Axis:= _stAXIS_REF, Execute:= FALSE, Position:= FB_MC2_AxisBasic_M_nMC_SetPositionRelative_lrPosition, Mode:= TRUE); 
		
